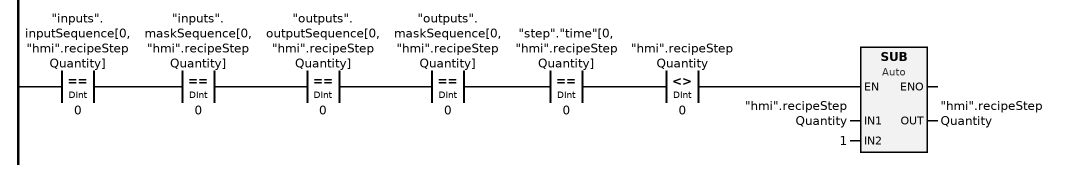
   RUNG wire#powerrail
      { S7_Templates := "SrcType := DInt" } NE_Contact(in1 := "inputs".inputSequence[0, 25], in2 := 0)
      wire#w1
      Move(in := 25, out1 => "hmi".recipeStepQuantity)
   END_RUNG
   RUNG wire#powerrail
      { S7_Templates := "SrcType := DInt" } NE_Contact(in1 := "inputs".maskSequence[0, 25], in2 := 0)
   END_RUNG wire#w1
   RUNG wire#powerrail
      { S7_Templates := "SrcType := DInt" } NE_Contact(in1 := "outputs".outputSequence[0, 25], in2 := 0)
   END_RUNG wire#w1
   RUNG wire#powerrail
      { S7_Templates := "SrcType := DInt" } NE_Contact(in1 := "outputs".maskSequence[0, 25], in2 := 0)
   END_RUNG wire#w1
   RUNG wire#powerrail
      { S7_Templates := "SrcType := DInt" } NE_Contact(in1 := "step"."time"[0, 25], in2 := 0)
   END_RUNG wire#w1
   RUNG wire#powerrail
      { S7_Templates := "SrcType := DInt" } LT_Contact(in1 := "hmi".recipeStepQuantity, in2 := 25)
      wire#w2
      { S7_Templates := "SrcType := DInt" } NE_Contact(in1 := "inputs".inputSequence[0, 24], in2 := 0)
      wire#w3
      Move(in := 24, out1 => "hmi".recipeStepQuantity)
   END_RUNG
   RUNG wire#w2
      { S7_Templates := "SrcType := DInt" } NE_Contact(in1 := "inputs".maskSequence[0, 24], in2 := 0)
   END_RUNG wire#w3
   RUNG wire#w2
      { S7_Templates := "SrcType := DInt" } NE_Contact(in1 := "outputs".outputSequence[0, 24], in2 := 0)
   END_RUNG wire#w3
   RUNG wire#w2
      { S7_Templates := "SrcType := DInt" } NE_Contact(in1 := "outputs".maskSequence[0, 24], in2 := 0)
   END_RUNG wire#w3
   RUNG wire#w2
      { S7_Templates := "SrcType := DInt" } NE_Contact(in1 := "step"."time"[0, 24], in2 := 0)
   END_RUNG wire#w3
   RUNG wire#powerrail
      { S7_Templates := "SrcType := DInt" } LT_Contact(in1 := "hmi".recipeStepQuantity, in2 := 24)
      wire#w4
      { S7_Templates := "SrcType := DInt" } NE_Contact(in1 := "inputs".inputSequence[0, 23], in2 := 0)
      wire#w5
      Move(in := 23, out1 => "hmi".recipeStepQuantity)
   END_RUNG
   RUNG wire#w4
      { S7_Templates := "SrcType := DInt" } NE_Contact(in1 := "inputs".maskSequence[0, 23], in2 := 0)
   END_RUNG wire#w5
   RUNG wire#w4
      { S7_Templates := "SrcType := DInt" } NE_Contact(in1 := "outputs".outputSequence[0, 23], in2 := 0)
   END_RUNG wire#w5
   RUNG wire#w4
      { S7_Templates := "SrcType := DInt" } NE_Contact(in1 := "outputs".maskSequence[0, 23], in2 := 0)
   END_RUNG wire#w5
   RUNG wire#w4
      { S7_Templates := "SrcType := DInt" } NE_Contact(in1 := "step"."time"[0, 23], in2 := 0)
   END_RUNG wire#w5
   RUNG wire#powerrail
      { S7_Templates := "SrcType := DInt" } LT_Contact(in1 := "hmi".recipeStepQuantity, in2 := 23)
      wire#w6
      { S7_Templates := "SrcType := DInt" } NE_Contact(in1 := "inputs".inputSequence[0, 22], in2 := 0)
      wire#w7
      Move(in := 22, out1 => "hmi".recipeStepQuantity)
   END_RUNG
   RUNG wire#w6
      { S7_Templates := "SrcType := DInt" } NE_Contact(in1 := "inputs".maskSequence[0, 22], in2 := 0)
   END_RUNG wire#w7
   RUNG wire#w6
      { S7_Templates := "SrcType := DInt" } NE_Contact(in1 := "outputs".outputSequence[0, 22], in2 := 0)
   END_RUNG wire#w7
   RUNG wire#w6
      { S7_Templates := "SrcType := DInt" } NE_Contact(in1 := "outputs".maskSequence[0, 22], in2 := 0)
   END_RUNG wire#w7
   RUNG wire#w6
      { S7_Templates := "SrcType := DInt" } NE_Contact(in1 := "step"."time"[0, 22], in2 := 0)
   END_RUNG wire#w7
   RUNG wire#powerrail
      { S7_Templates := "SrcType := DInt" } LT_Contact(in1 := "hmi".recipeStepQuantity, in2 := 22)
      wire#w8
      { S7_Templates := "SrcType := DInt" } NE_Contact(in1 := "inputs".inputSequence[0, 21], in2 := 0)
      wire#w9
      Move(in := 21, out1 => "hmi".recipeStepQuantity)
   END_RUNG
   RUNG wire#w8
      { S7_Templates := "SrcType := DInt" } NE_Contact(in1 := "inputs".maskSequence[0, 21], in2 := 0)
   END_RUNG wire#w9
   RUNG wire#w8
      { S7_Templates := "SrcType := DInt" } NE_Contact(in1 := "outputs".outputSequence[0, 21], in2 := 0)
   END_RUNG wire#w9
   RUNG wire#w8
      { S7_Templates := "SrcType := DInt" } NE_Contact(in1 := "outputs".maskSequence[0, 21], in2 := 0)
   END_RUNG wire#w9
   RUNG wire#w8
      { S7_Templates := "SrcType := DInt" } NE_Contact(in1 := "step"."time"[0, 21], in2 := 0)
   END_RUNG wire#w9
   RUNG wire#powerrail
      { S7_Templates := "SrcType := DInt" } LT_Contact(in1 := "hmi".recipeStepQuantity, in2 := 21)
      wire#w10
      { S7_Templates := "SrcType := DInt" } NE_Contact(in1 := "inputs".inputSequence[0, 20], in2 := 0)
      wire#w11
      Move(in := 20, out1 => "hmi".recipeStepQuantity)
   END_RUNG
   RUNG wire#w10
      { S7_Templates := "SrcType := DInt" } NE_Contact(in1 := "inputs".maskSequence[0, 20], in2 := 0)
   END_RUNG wire#w11
   RUNG wire#w10
      { S7_Templates := "SrcType := DInt" } NE_Contact(in1 := "outputs".outputSequence[0, 20], in2 := 0)
   END_RUNG wire#w11
   RUNG wire#w10
      { S7_Templates := "SrcType := DInt" } NE_Contact(in1 := "outputs".maskSequence[0, 20], in2 := 0)
   END_RUNG wire#w11
   RUNG wire#w10
      { S7_Templates := "SrcType := DInt" } NE_Contact(in1 := "step"."time"[0, 20], in2 := 0)
   END_RUNG wire#w11
   RUNG wire#powerrail
      { S7_Templates := "SrcType := DInt" } LT_Contact(in1 := "hmi".recipeStepQuantity, in2 := 20)
      wire#w12
      { S7_Templates := "SrcType := DInt" } NE_Contact(in1 := "inputs".inputSequence[0, 19], in2 := 0)
      wire#w13
      Move(in := 19, out1 => "hmi".recipeStepQuantity)
   END_RUNG
   RUNG wire#w12
      { S7_Templates := "SrcType := DInt" } NE_Contact(in1 := "inputs".maskSequence[0, 19], in2 := 0)
   END_RUNG wire#w13
   RUNG wire#w12
      { S7_Templates := "SrcType := DInt" } NE_Contact(in1 := "outputs".outputSequence[0, 19], in2 := 0)
   END_RUNG wire#w13
   RUNG wire#w12
      { S7_Templates := "SrcType := DInt" } NE_Contact(in1 := "outputs".maskSequence[0, 19], in2 := 0)
   END_RUNG wire#w13
   RUNG wire#w12
      { S7_Templates := "SrcType := DInt" } NE_Contact(in1 := "step"."time"[0, 19], in2 := 0)
   END_RUNG wire#w13
   RUNG wire#powerrail
      { S7_Templates := "SrcType := DInt" } LT_Contact(in1 := "hmi".recipeStepQuantity, in2 := 19)
      wire#w14
      { S7_Templates := "SrcType := DInt" } NE_Contact(in1 := "inputs".inputSequence[0, 18], in2 := 0)
      wire#w15
      Move(in := 18, out1 => "hmi".recipeStepQuantity)
   END_RUNG
   RUNG wire#w14
      { S7_Templates := "SrcType := DInt" } NE_Contact(in1 := "inputs".maskSequence[0, 18], in2 := 0)
   END_RUNG wire#w15
   RUNG wire#w14
      { S7_Templates := "SrcType := DInt" } NE_Contact(in1 := "outputs".outputSequence[0, 18], in2 := 0)
   END_RUNG wire#w15
   RUNG wire#w14
      { S7_Templates := "SrcType := DInt" } NE_Contact(in1 := "outputs".maskSequence[0, 18], in2 := 0)
   END_RUNG wire#w15
   RUNG wire#w14
      { S7_Templates := "SrcType := DInt" } NE_Contact(in1 := "step"."time"[0, 18], in2 := 0)
   END_RUNG wire#w15
   RUNG wire#powerrail
      { S7_Templates := "SrcType := DInt" } LT_Contact(in1 := "hmi".recipeStepQuantity, in2 := 18)
      wire#w16
      { S7_Templates := "SrcType := DInt" } NE_Contact(in1 := "inputs".inputSequence[0, 17], in2 := 0)
      wire#w17
      Move(in := 17, out1 => "hmi".recipeStepQuantity)
   END_RUNG
   RUNG wire#w16
      { S7_Templates := "SrcType := DInt" } NE_Contact(in1 := "inputs".maskSequence[0, 17], in2 := 0)
   END_RUNG wire#w17
   RUNG wire#w16
      { S7_Templates := "SrcType := DInt" } NE_Contact(in1 := "outputs".outputSequence[0, 17], in2 := 0)
   END_RUNG wire#w17
   RUNG wire#w16
      { S7_Templates := "SrcType := DInt" } NE_Contact(in1 := "outputs".maskSequence[0, 17], in2 := 0)
   END_RUNG wire#w17
   RUNG wire#w16
      { S7_Templates := "SrcType := DInt" } NE_Contact(in1 := "step"."time"[0, 17], in2 := 0)
   END_RUNG wire#w17
   RUNG wire#powerrail
      { S7_Templates := "SrcType := DInt" } LT_Contact(in1 := "hmi".recipeStepQuantity, in2 := 17)
      wire#w18
      { S7_Templates := "SrcType := DInt" } NE_Contact(in1 := "inputs".inputSequence[0, 16], in2 := 0)
      wire#w19
      Move(in := 16, out1 => "hmi".recipeStepQuantity)
   END_RUNG
   RUNG wire#w18
      { S7_Templates := "SrcType := DInt" } NE_Contact(in1 := "inputs".maskSequence[0, 16], in2 := 0)
   END_RUNG wire#w19
   RUNG wire#w18
      { S7_Templates := "SrcType := DInt" } NE_Contact(in1 := "outputs".outputSequence[0, 16], in2 := 0)
   END_RUNG wire#w19
   RUNG wire#w18
      { S7_Templates := "SrcType := DInt" } NE_Contact(in1 := "outputs".maskSequence[0, 16], in2 := 0)
   END_RUNG wire#w19
   RUNG wire#w18
      { S7_Templates := "SrcType := DInt" } NE_Contact(in1 := "step"."time"[0, 16], in2 := 0)
   END_RUNG wire#w19
   RUNG wire#powerrail
      { S7_Templates := "SrcType := DInt" } LT_Contact(in1 := "hmi".recipeStepQuantity, in2 := 16)
      wire#w20
      { S7_Templates := "SrcType := DInt" } NE_Contact(in1 := "inputs".inputSequence[0, 15], in2 := 0)
      wire#w21
      Move(in := 15, out1 => "hmi".recipeStepQuantity)
   END_RUNG
   RUNG wire#w20
      { S7_Templates := "SrcType := DInt" } NE_Contact(in1 := "inputs".maskSequence[0, 15], in2 := 0)
   END_RUNG wire#w21
   RUNG wire#w20
      { S7_Templates := "SrcType := DInt" } NE_Contact(in1 := "outputs".outputSequence[0, 15], in2 := 0)
   END_RUNG wire#w21
   RUNG wire#w20
      { S7_Templates := "SrcType := DInt" } NE_Contact(in1 := "outputs".maskSequence[0, 15], in2 := 0)
   END_RUNG wire#w21
   RUNG wire#w20
      { S7_Templates := "SrcType := DInt" } NE_Contact(in1 := "step"."time"[0, 15], in2 := 0)
   END_RUNG wire#w21
   RUNG wire#powerrail
      { S7_Templates := "SrcType := DInt" } LT_Contact(in1 := "hmi".recipeStepQuantity, in2 := 15)
      wire#w22
      { S7_Templates := "SrcType := DInt" } NE_Contact(in1 := "inputs".inputSequence[0, 14], in2 := 0)
      wire#w23
      Move(in := 14, out1 => "hmi".recipeStepQuantity)
   END_RUNG
   RUNG wire#w22
      { S7_Templates := "SrcType := DInt" } NE_Contact(in1 := "inputs".maskSequence[0, 14], in2 := 0)
   END_RUNG wire#w23
   RUNG wire#w22
      { S7_Templates := "SrcType := DInt" } NE_Contact(in1 := "outputs".outputSequence[0, 14], in2 := 0)
   END_RUNG wire#w23
   RUNG wire#w22
      { S7_Templates := "SrcType := DInt" } NE_Contact(in1 := "outputs".maskSequence[0, 14], in2 := 0)
   END_RUNG wire#w23
   RUNG wire#w22
      { S7_Templates := "SrcType := DInt" } NE_Contact(in1 := "step"."time"[0, 14], in2 := 0)
   END_RUNG wire#w23
   RUNG wire#powerrail
      { S7_Templates := "SrcType := DInt" } LT_Contact(in1 := "hmi".recipeStepQuantity, in2 := 14)
      wire#w24
      { S7_Templates := "SrcType := DInt" } NE_Contact(in1 := "inputs".inputSequence[0, 13], in2 := 0)
      wire#w25
      Move(in := 13, out1 => "hmi".recipeStepQuantity)
   END_RUNG
   RUNG wire#w24
      { S7_Templates := "SrcType := DInt" } NE_Contact(in1 := "inputs".maskSequence[0, 13], in2 := 0)
   END_RUNG wire#w25
   RUNG wire#w24
      { S7_Templates := "SrcType := DInt" } NE_Contact(in1 := "outputs".outputSequence[0, 13], in2 := 0)
   END_RUNG wire#w25
   RUNG wire#w24
      { S7_Templates := "SrcType := DInt" } NE_Contact(in1 := "outputs".maskSequence[0, 13], in2 := 0)
   END_RUNG wire#w25
   RUNG wire#w24
      { S7_Templates := "SrcType := DInt" } NE_Contact(in1 := "step"."time"[0, 13], in2 := 0)
   END_RUNG wire#w25
   RUNG wire#powerrail
      { S7_Templates := "SrcType := DInt" } LT_Contact(in1 := "hmi".recipeStepQuantity, in2 := 13)
      wire#w26
      { S7_Templates := "SrcType := DInt" } NE_Contact(in1 := "inputs".inputSequence[0, 12], in2 := 0)
      wire#w27
      Move(in := 12, out1 => "hmi".recipeStepQuantity)
   END_RUNG
   RUNG wire#w26
      { S7_Templates := "SrcType := DInt" } NE_Contact(in1 := "inputs".maskSequence[0, 12], in2 := 0)
   END_RUNG wire#w27
   RUNG wire#w26
      { S7_Templates := "SrcType := DInt" } NE_Contact(in1 := "outputs".outputSequence[0, 12], in2 := 0)
   END_RUNG wire#w27
   RUNG wire#w26
      { S7_Templates := "SrcType := DInt" } NE_Contact(in1 := "outputs".maskSequence[0, 12], in2 := 0)
   END_RUNG wire#w27
   RUNG wire#w26
      { S7_Templates := "SrcType := DInt" } NE_Contact(in1 := "step"."time"[0, 12], in2 := 0)
   END_RUNG wire#w27
   RUNG wire#powerrail
      { S7_Templates := "SrcType := DInt" } LT_Contact(in1 := "hmi".recipeStepQuantity, in2 := 12)
      wire#w28
      { S7_Templates := "SrcType := DInt" } NE_Contact(in1 := "inputs".inputSequence[0, 11], in2 := 0)
      wire#w29
      Move(in := 11, out1 => "hmi".recipeStepQuantity)
   END_RUNG
   RUNG wire#w28
      { S7_Templates := "SrcType := DInt" } NE_Contact(in1 := "inputs".maskSequence[0, 11], in2 := 0)
   END_RUNG wire#w29
   RUNG wire#w28
      { S7_Templates := "SrcType := DInt" } NE_Contact(in1 := "outputs".outputSequence[0, 11], in2 := 0)
   END_RUNG wire#w29
   RUNG wire#w28
      { S7_Templates := "SrcType := DInt" } NE_Contact(in1 := "outputs".maskSequence[0, 11], in2 := 0)
   END_RUNG wire#w29
   RUNG wire#w28
      { S7_Templates := "SrcType := DInt" } NE_Contact(in1 := "step"."time"[0, 11], in2 := 0)
   END_RUNG wire#w29
   RUNG wire#powerrail
      { S7_Templates := "SrcType := DInt" } LT_Contact(in1 := "hmi".recipeStepQuantity, in2 := 11)
      wire#w30
      { S7_Templates := "SrcType := DInt" } NE_Contact(in1 := "inputs".inputSequence[0, 10], in2 := 0)
      wire#w31
      Move(in := 10, out1 => "hmi".recipeStepQuantity)
   END_RUNG
   RUNG wire#w30
      { S7_Templates := "SrcType := DInt" } NE_Contact(in1 := "inputs".maskSequence[0, 10], in2 := 0)
   END_RUNG wire#w31
   RUNG wire#w30
      { S7_Templates := "SrcType := DInt" } NE_Contact(in1 := "outputs".outputSequence[0, 10], in2 := 0)
   END_RUNG wire#w31
   RUNG wire#w30
      { S7_Templates := "SrcType := DInt" } NE_Contact(in1 := "outputs".maskSequence[0, 10], in2 := 0)
   END_RUNG wire#w31
   RUNG wire#w30
      { S7_Templates := "SrcType := DInt" } NE_Contact(in1 := "step"."time"[0, 10], in2 := 0)
   END_RUNG wire#w31
   RUNG wire#powerrail
      { S7_Templates := "SrcType := DInt" } LT_Contact(in1 := "hmi".recipeStepQuantity, in2 := 10)
      wire#w32
      { S7_Templates := "SrcType := DInt" } NE_Contact(in1 := "inputs".inputSequence[0, 9], in2 := 0)
      wire#w33
      Move(in := 9, out1 => "hmi".recipeStepQuantity)
   END_RUNG
   RUNG wire#w32
      { S7_Templates := "SrcType := DInt" } NE_Contact(in1 := "inputs".maskSequence[0, 9], in2 := 0)
   END_RUNG wire#w33
   RUNG wire#w32
      { S7_Templates := "SrcType := DInt" } NE_Contact(in1 := "outputs".outputSequence[0, 9], in2 := 0)
   END_RUNG wire#w33
   RUNG wire#w32
      { S7_Templates := "SrcType := DInt" } NE_Contact(in1 := "outputs".maskSequence[0, 9], in2 := 0)
   END_RUNG wire#w33
   RUNG wire#w32
      { S7_Templates := "SrcType := DInt" } NE_Contact(in1 := "step"."time"[0, 9], in2 := 0)
   END_RUNG wire#w33
   RUNG wire#powerrail
      { S7_Templates := "SrcType := DInt" } LT_Contact(in1 := "hmi".recipeStepQuantity, in2 := 9)
      wire#w34
      { S7_Templates := "SrcType := DInt" } NE_Contact(in1 := "inputs".inputSequence[0, 8], in2 := 0)
      wire#w35
      Move(in := 8, out1 => "hmi".recipeStepQuantity)
   END_RUNG
   RUNG wire#w34
      { S7_Templates := "SrcType := DInt" } NE_Contact(in1 := "inputs".maskSequence[0, 8], in2 := 0)
   END_RUNG wire#w35
   RUNG wire#w34
      { S7_Templates := "SrcType := DInt" } NE_Contact(in1 := "outputs".outputSequence[0, 8], in2 := 0)
   END_RUNG wire#w35
   RUNG wire#w34
      { S7_Templates := "SrcType := DInt" } NE_Contact(in1 := "outputs".maskSequence[0, 8], in2 := 0)
   END_RUNG wire#w35
   RUNG wire#w34
      { S7_Templates := "SrcType := DInt" } NE_Contact(in1 := "step"."time"[0, 8], in2 := 0)
   END_RUNG wire#w35
   RUNG wire#powerrail
      { S7_Templates := "SrcType := DInt" } LT_Contact(in1 := "hmi".recipeStepQuantity, in2 := 8)
      wire#w36
      { S7_Templates := "SrcType := DInt" } NE_Contact(in1 := "inputs".inputSequence[0, 7], in2 := 0)
      wire#w37
      Move(in := 7, out1 => "hmi".recipeStepQuantity)
   END_RUNG
   RUNG wire#w36
      { S7_Templates := "SrcType := DInt" } NE_Contact(in1 := "inputs".maskSequence[0, 7], in2 := 0)
   END_RUNG wire#w37
   RUNG wire#w36
      { S7_Templates := "SrcType := DInt" } NE_Contact(in1 := "outputs".outputSequence[0, 7], in2 := 0)
   END_RUNG wire#w37
   RUNG wire#w36
      { S7_Templates := "SrcType := DInt" } NE_Contact(in1 := "outputs".maskSequence[0, 7], in2 := 0)
   END_RUNG wire#w37
   RUNG wire#w36
      { S7_Templates := "SrcType := DInt" } NE_Contact(in1 := "step"."time"[0, 7], in2 := 0)
   END_RUNG wire#w37
   RUNG wire#powerrail
      { S7_Templates := "SrcType := DInt" } LT_Contact(in1 := "hmi".recipeStepQuantity, in2 := 7)
      wire#w38
      { S7_Templates := "SrcType := DInt" } NE_Contact(in1 := "inputs".inputSequence[0, 6], in2 := 0)
      wire#w39
      Move(in := 6, out1 => "hmi".recipeStepQuantity)
   END_RUNG
   RUNG wire#w38
      { S7_Templates := "SrcType := DInt" } NE_Contact(in1 := "inputs".maskSequence[0, 6], in2 := 0)
   END_RUNG wire#w39
   RUNG wire#w38
      { S7_Templates := "SrcType := DInt" } NE_Contact(in1 := "outputs".outputSequence[0, 6], in2 := 0)
   END_RUNG wire#w39
   RUNG wire#w38
      { S7_Templates := "SrcType := DInt" } NE_Contact(in1 := "outputs".maskSequence[0, 6], in2 := 0)
   END_RUNG wire#w39
   RUNG wire#w38
      { S7_Templates := "SrcType := DInt" } NE_Contact(in1 := "step"."time"[0, 6], in2 := 0)
   END_RUNG wire#w39
   RUNG wire#powerrail
      { S7_Templates := "SrcType := DInt" } LT_Contact(in1 := "hmi".recipeStepQuantity, in2 := 6)
      wire#w40
      { S7_Templates := "SrcType := DInt" } NE_Contact(in1 := "inputs".inputSequence[0, 5], in2 := 0)
      wire#w41
      Move(in := 5, out1 => "hmi".recipeStepQuantity)
   END_RUNG
   RUNG wire#w40
      { S7_Templates := "SrcType := DInt" } NE_Contact(in1 := "inputs".maskSequence[0, 5], in2 := 0)
   END_RUNG wire#w41
   RUNG wire#w40
      { S7_Templates := "SrcType := DInt" } NE_Contact(in1 := "outputs".outputSequence[0, 5], in2 := 0)
   END_RUNG wire#w41
   RUNG wire#w40
      { S7_Templates := "SrcType := DInt" } NE_Contact(in1 := "outputs".maskSequence[0, 5], in2 := 0)
   END_RUNG wire#w41
   RUNG wire#w40
      { S7_Templates := "SrcType := DInt" } NE_Contact(in1 := "step"."time"[0, 5], in2 := 0)
   END_RUNG wire#w41
   RUNG wire#powerrail
      { S7_Templates := "SrcType := DInt" } LT_Contact(in1 := "hmi".recipeStepQuantity, in2 := 5)
      wire#w42
      { S7_Templates := "SrcType := DInt" } NE_Contact(in1 := "inputs".inputSequence[0, 4], in2 := 0)
      wire#w43
      Move(in := 4, out1 => "hmi".recipeStepQuantity)
   END_RUNG
   RUNG wire#w42
      { S7_Templates := "SrcType := DInt" } NE_Contact(in1 := "inputs".maskSequence[0, 4], in2 := 0)
   END_RUNG wire#w43
   RUNG wire#w42
      { S7_Templates := "SrcType := DInt" } NE_Contact(in1 := "outputs".outputSequence[0, 4], in2 := 0)
   END_RUNG wire#w43
   RUNG wire#w42
      { S7_Templates := "SrcType := DInt" } NE_Contact(in1 := "outputs".maskSequence[0, 4], in2 := 0)
   END_RUNG wire#w43
   RUNG wire#w42
      { S7_Templates := "SrcType := DInt" } NE_Contact(in1 := "step"."time"[0, 4], in2 := 0)
   END_RUNG wire#w43
   RUNG wire#powerrail
      { S7_Templates := "SrcType := DInt" } LT_Contact(in1 := "hmi".recipeStepQuantity, in2 := 4)
      wire#w44
      { S7_Templates := "SrcType := DInt" } NE_Contact(in1 := "inputs".inputSequence[0, 3], in2 := 0)
      wire#w45
      Move(in := 3, out1 => "hmi".recipeStepQuantity)
   END_RUNG
   RUNG wire#w44
      { S7_Templates := "SrcType := DInt" } NE_Contact(in1 := "inputs".maskSequence[0, 3], in2 := 0)
   END_RUNG wire#w45
   RUNG wire#w44
      { S7_Templates := "SrcType := DInt" } NE_Contact(in1 := "outputs".outputSequence[0, 3], in2 := 0)
   END_RUNG wire#w45
   RUNG wire#w44
      { S7_Templates := "SrcType := DInt" } NE_Contact(in1 := "outputs".maskSequence[0, 3], in2 := 0)
   END_RUNG wire#w45
   RUNG wire#w44
      { S7_Templates := "SrcType := DInt" } NE_Contact(in1 := "step"."time"[0, 3], in2 := 0)
   END_RUNG wire#w45
   RUNG wire#powerrail
      { S7_Templates := "SrcType := DInt" } LT_Contact(in1 := "hmi".recipeStepQuantity, in2 := 3)
      wire#w46
      { S7_Templates := "SrcType := DInt" } NE_Contact(in1 := "inputs".inputSequence[0, 2], in2 := 0)
      wire#w47
      Move(in := 2, out1 => "hmi".recipeStepQuantity)
   END_RUNG
   RUNG wire#w46
      { S7_Templates := "SrcType := DInt" } NE_Contact(in1 := "inputs".maskSequence[0, 2], in2 := 0)
   END_RUNG wire#w47
   RUNG wire#w46
      { S7_Templates := "SrcType := DInt" } NE_Contact(in1 := "outputs".outputSequence[0, 2], in2 := 0)
   END_RUNG wire#w47
   RUNG wire#w46
      { S7_Templates := "SrcType := DInt" } NE_Contact(in1 := "outputs".maskSequence[0, 2], in2 := 0)
   END_RUNG wire#w47
   RUNG wire#w46
      { S7_Templates := "SrcType := DInt" } NE_Contact(in1 := "step"."time"[0, 2], in2 := 0)
   END_RUNG wire#w47
   RUNG wire#powerrail
      { S7_Templates := "SrcType := DInt" } LT_Contact(in1 := "hmi".recipeStepQuantity, in2 := 2)
      wire#w48
      { S7_Templates := "SrcType := DInt" } NE_Contact(in1 := "inputs".inputSequence[0, 1], in2 := 0)
      wire#w49
      Move(in := 1, out1 => "hmi".recipeStepQuantity)
   END_RUNG
   RUNG wire#w48
      { S7_Templates := "SrcType := DInt" } NE_Contact(in1 := "inputs".maskSequence[0, 1], in2 := 0)
   END_RUNG wire#w49
   RUNG wire#w48
      { S7_Templates := "SrcType := DInt" } NE_Contact(in1 := "outputs".outputSequence[0, 1], in2 := 0)
   END_RUNG wire#w49
   RUNG wire#w48
      { S7_Templates := "SrcType := DInt" } NE_Contact(in1 := "outputs".maskSequence[0, 1], in2 := 0)
   END_RUNG wire#w49
   RUNG wire#w48
      { S7_Templates := "SrcType := DInt" } NE_Contact(in1 := "step"."time"[0, 1], in2 := 0)
   END_RUNG wire#w49
   RUNG wire#powerrail
      { S7_Templates := "SrcType := DInt" } LT_Contact(in1 := "hmi".recipeStepQuantity, in2 := 1)
      Move(in := 0, out1 => "hmi".recipeStepQuantity)
   END_RUNG
   RUNG wire#powerrail
      { S7_Templates := "SrcType := DInt" } EQ_Contact(in1 := "inputs".inputSequence[0, "hmi".recipeStepQuantity], in2 := 0)
      { S7_Templates := "SrcType := DInt" } EQ_Contact(in1 := "inputs".maskSequence[0, "hmi".recipeStepQuantity], in2 := 0)
      { S7_Templates := "SrcType := DInt" } EQ_Contact(in1 := "outputs".outputSequence[0, "hmi".recipeStepQuantity], in2 := 0)
      { S7_Templates := "SrcType := DInt" } EQ_Contact(in1 := "outputs".maskSequence[0, "hmi".recipeStepQuantity], in2 := 0)
      { S7_Templates := "SrcType := DInt" } EQ_Contact(in1 := "step"."time"[0, "hmi".recipeStepQuantity], in2 := 0)
      { S7_Templates := "SrcType := DInt" } NE_Contact(in1 := "hmi".recipeStepQuantity, in2 := 0)
      Sub(in1 := "hmi".recipeStepQuantity, in2 := 1, out => "hmi".recipeStepQuantity)
   END_RUNG
   // the same network as SCL:
   IF ("inputs".inputSequence[0, 25] <> 0) OR ("inputs".maskSequence[0, 25] <> 0) OR ("outputs".outputSequence[0, 25] <> 0) OR ("outputs".maskSequence[0, 25] <> 0) OR ("step"."time"[0, 25] <> 0) THEN
       "hmi".recipeStepQuantity := 25;
   END_IF;
   IF ("hmi".recipeStepQuantity < 25) AND (("inputs".inputSequence[0, 24] <> 0) OR ("inputs".maskSequence[0, 24] <> 0) OR ("outputs".outputSequence[0, 24] <> 0) OR ("outputs".maskSequence[0, 24] <> 0) OR ("step"."time"[0, 24] <> 0)) THEN
       "hmi".recipeStepQuantity := 24;
   END_IF;
   IF ("hmi".recipeStepQuantity < 24) AND (("inputs".inputSequence[0, 23] <> 0) OR ("inputs".maskSequence[0, 23] <> 0) OR ("outputs".outputSequence[0, 23] <> 0) OR ("outputs".maskSequence[0, 23] <> 0) OR ("step"."time"[0, 23] <> 0)) THEN
       "hmi".recipeStepQuantity := 23;
   END_IF;
   IF ("hmi".recipeStepQuantity < 23) AND (("inputs".inputSequence[0, 22] <> 0) OR ("inputs".maskSequence[0, 22] <> 0) OR ("outputs".outputSequence[0, 22] <> 0) OR ("outputs".maskSequence[0, 22] <> 0) OR ("step"."time"[0, 22] <> 0)) THEN
       "hmi".recipeStepQuantity := 22;
   END_IF;
   IF ("hmi".recipeStepQuantity < 22) AND (("inputs".inputSequence[0, 21] <> 0) OR ("inputs".maskSequence[0, 21] <> 0) OR ("outputs".outputSequence[0, 21] <> 0) OR ("outputs".maskSequence[0, 21] <> 0) OR ("step"."time"[0, 21] <> 0)) THEN
       "hmi".recipeStepQuantity := 21;
   END_IF;
   IF ("hmi".recipeStepQuantity < 21) AND (("inputs".inputSequence[0, 20] <> 0) OR ("inputs".maskSequence[0, 20] <> 0) OR ("outputs".outputSequence[0, 20] <> 0) OR ("outputs".maskSequence[0, 20] <> 0) OR ("step"."time"[0, 20] <> 0)) THEN
       "hmi".recipeStepQuantity := 20;
   END_IF;
   IF ("hmi".recipeStepQuantity < 20) AND (("inputs".inputSequence[0, 19] <> 0) OR ("inputs".maskSequence[0, 19] <> 0) OR ("outputs".outputSequence[0, 19] <> 0) OR ("outputs".maskSequence[0, 19] <> 0) OR ("step"."time"[0, 19] <> 0)) THEN
       "hmi".recipeStepQuantity := 19;
   END_IF;
   IF ("hmi".recipeStepQuantity < 19) AND (("inputs".inputSequence[0, 18] <> 0) OR ("inputs".maskSequence[0, 18] <> 0) OR ("outputs".outputSequence[0, 18] <> 0) OR ("outputs".maskSequence[0, 18] <> 0) OR ("step"."time"[0, 18] <> 0)) THEN
       "hmi".recipeStepQuantity := 18;
   END_IF;
   IF ("hmi".recipeStepQuantity < 18) AND (("inputs".inputSequence[0, 17] <> 0) OR ("inputs".maskSequence[0, 17] <> 0) OR ("outputs".outputSequence[0, 17] <> 0) OR ("outputs".maskSequence[0, 17] <> 0) OR ("step"."time"[0, 17] <> 0)) THEN
       "hmi".recipeStepQuantity := 17;
   END_IF;
   IF ("hmi".recipeStepQuantity < 17) AND (("inputs".inputSequence[0, 16] <> 0) OR ("inputs".maskSequence[0, 16] <> 0) OR ("outputs".outputSequence[0, 16] <> 0) OR ("outputs".maskSequence[0, 16] <> 0) OR ("step"."time"[0, 16] <> 0)) THEN
       "hmi".recipeStepQuantity := 16;
   END_IF;
   IF ("hmi".recipeStepQuantity < 16) AND (("inputs".inputSequence[0, 15] <> 0) OR ("inputs".maskSequence[0, 15] <> 0) OR ("outputs".outputSequence[0, 15] <> 0) OR ("outputs".maskSequence[0, 15] <> 0) OR ("step"."time"[0, 15] <> 0)) THEN
       "hmi".recipeStepQuantity := 15;
   END_IF;
   IF ("hmi".recipeStepQuantity < 15) AND (("inputs".inputSequence[0, 14] <> 0) OR ("inputs".maskSequence[0, 14] <> 0) OR ("outputs".outputSequence[0, 14] <> 0) OR ("outputs".maskSequence[0, 14] <> 0) OR ("step"."time"[0, 14] <> 0)) THEN
       "hmi".recipeStepQuantity := 14;
   END_IF;
   IF ("hmi".recipeStepQuantity < 14) AND (("inputs".inputSequence[0, 13] <> 0) OR ("inputs".maskSequence[0, 13] <> 0) OR ("outputs".outputSequence[0, 13] <> 0) OR ("outputs".maskSequence[0, 13] <> 0) OR ("step"."time"[0, 13] <> 0)) THEN
       "hmi".recipeStepQuantity := 13;
   END_IF;
   IF ("hmi".recipeStepQuantity < 13) AND (("inputs".inputSequence[0, 12] <> 0) OR ("inputs".maskSequence[0, 12] <> 0) OR ("outputs".outputSequence[0, 12] <> 0) OR ("outputs".maskSequence[0, 12] <> 0) OR ("step"."time"[0, 12] <> 0)) THEN
       "hmi".recipeStepQuantity := 12;
   END_IF;
   IF ("hmi".recipeStepQuantity < 12) AND (("inputs".inputSequence[0, 11] <> 0) OR ("inputs".maskSequence[0, 11] <> 0) OR ("outputs".outputSequence[0, 11] <> 0) OR ("outputs".maskSequence[0, 11] <> 0) OR ("step"."time"[0, 11] <> 0)) THEN
       "hmi".recipeStepQuantity := 11;
   END_IF;
   IF ("hmi".recipeStepQuantity < 11) AND (("inputs".inputSequence[0, 10] <> 0) OR ("inputs".maskSequence[0, 10] <> 0) OR ("outputs".outputSequence[0, 10] <> 0) OR ("outputs".maskSequence[0, 10] <> 0) OR ("step"."time"[0, 10] <> 0)) THEN
       "hmi".recipeStepQuantity := 10;
   END_IF;
   IF ("hmi".recipeStepQuantity < 10) AND (("inputs".inputSequence[0, 9] <> 0) OR ("inputs".maskSequence[0, 9] <> 0) OR ("outputs".outputSequence[0, 9] <> 0) OR ("outputs".maskSequence[0, 9] <> 0) OR ("step"."time"[0, 9] <> 0)) THEN
       "hmi".recipeStepQuantity := 9;
   END_IF;
   IF ("hmi".recipeStepQuantity < 9) AND (("inputs".inputSequence[0, 8] <> 0) OR ("inputs".maskSequence[0, 8] <> 0) OR ("outputs".outputSequence[0, 8] <> 0) OR ("outputs".maskSequence[0, 8] <> 0) OR ("step"."time"[0, 8] <> 0)) THEN
       "hmi".recipeStepQuantity := 8;
   END_IF;
   IF ("hmi".recipeStepQuantity < 8) AND (("inputs".inputSequence[0, 7] <> 0) OR ("inputs".maskSequence[0, 7] <> 0) OR ("outputs".outputSequence[0, 7] <> 0) OR ("outputs".maskSequence[0, 7] <> 0) OR ("step"."time"[0, 7] <> 0)) THEN
       "hmi".recipeStepQuantity := 7;
   END_IF;
   IF ("hmi".recipeStepQuantity < 7) AND (("inputs".inputSequence[0, 6] <> 0) OR ("inputs".maskSequence[0, 6] <> 0) OR ("outputs".outputSequence[0, 6] <> 0) OR ("outputs".maskSequence[0, 6] <> 0) OR ("step"."time"[0, 6] <> 0)) THEN
       "hmi".recipeStepQuantity := 6;
   END_IF;
   IF ("hmi".recipeStepQuantity < 6) AND (("inputs".inputSequence[0, 5] <> 0) OR ("inputs".maskSequence[0, 5] <> 0) OR ("outputs".outputSequence[0, 5] <> 0) OR ("outputs".maskSequence[0, 5] <> 0) OR ("step"."time"[0, 5] <> 0)) THEN
       "hmi".recipeStepQuantity := 5;
   END_IF;
   IF ("hmi".recipeStepQuantity < 5) AND (("inputs".inputSequence[0, 4] <> 0) OR ("inputs".maskSequence[0, 4] <> 0) OR ("outputs".outputSequence[0, 4] <> 0) OR ("outputs".maskSequence[0, 4] <> 0) OR ("step"."time"[0, 4] <> 0)) THEN
       "hmi".recipeStepQuantity := 4;
   END_IF;
   IF ("hmi".recipeStepQuantity < 4) AND (("inputs".inputSequence[0, 3] <> 0) OR ("inputs".maskSequence[0, 3] <> 0) OR ("outputs".outputSequence[0, 3] <> 0) OR ("outputs".maskSequence[0, 3] <> 0) OR ("step"."time"[0, 3] <> 0)) THEN
       "hmi".recipeStepQuantity := 3;
   END_IF;
   IF ("hmi".recipeStepQuantity < 3) AND (("inputs".inputSequence[0, 2] <> 0) OR ("inputs".maskSequence[0, 2] <> 0) OR ("outputs".outputSequence[0, 2] <> 0) OR ("outputs".maskSequence[0, 2] <> 0) OR ("step"."time"[0, 2] <> 0)) THEN
       "hmi".recipeStepQuantity := 2;
   END_IF;
   IF ("hmi".recipeStepQuantity < 2) AND (("inputs".inputSequence[0, 1] <> 0) OR ("inputs".maskSequence[0, 1] <> 0) OR ("outputs".outputSequence[0, 1] <> 0) OR ("outputs".maskSequence[0, 1] <> 0) OR ("step"."time"[0, 1] <> 0)) THEN
       "hmi".recipeStepQuantity := 1;
   END_IF;
   IF "hmi".recipeStepQuantity < 1 THEN "hmi".recipeStepQuantity := 0; END_IF;
   IF ("inputs".inputSequence[0, "hmi".recipeStepQuantity] = 0) AND ("inputs".maskSequence[0, "hmi".recipeStepQuantity] = 0) AND ("outputs".outputSequence[0, "hmi".recipeStepQuantity] = 0) AND ("outputs".maskSequence[0, "hmi".recipeStepQuantity] = 0) AND ("step"."time"[0, "hmi".recipeStepQuantity] = 0) AND ("hmi".recipeStepQuantity <> 0) THEN
       "hmi".recipeStepQuantity := "hmi".recipeStepQuantity - 1;
   END_IF;
END_REGION

REGION Network 9: INPUTS STATUS TO SHOW ON SCREEN
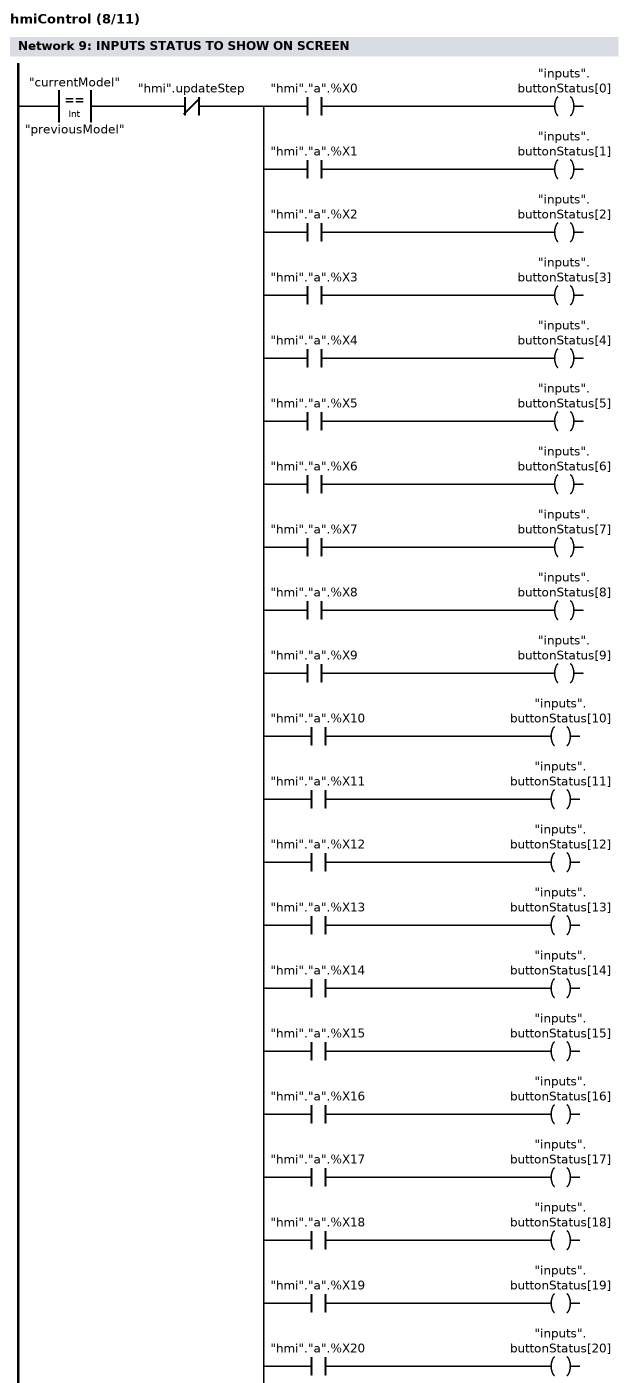
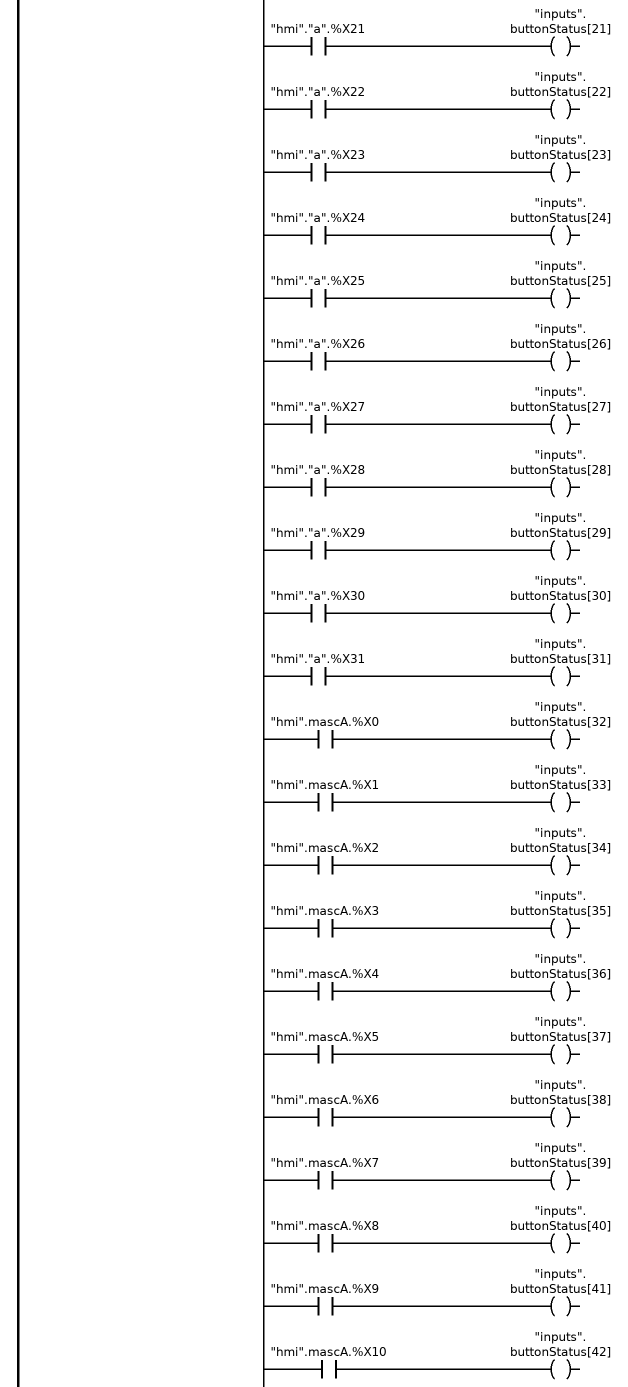
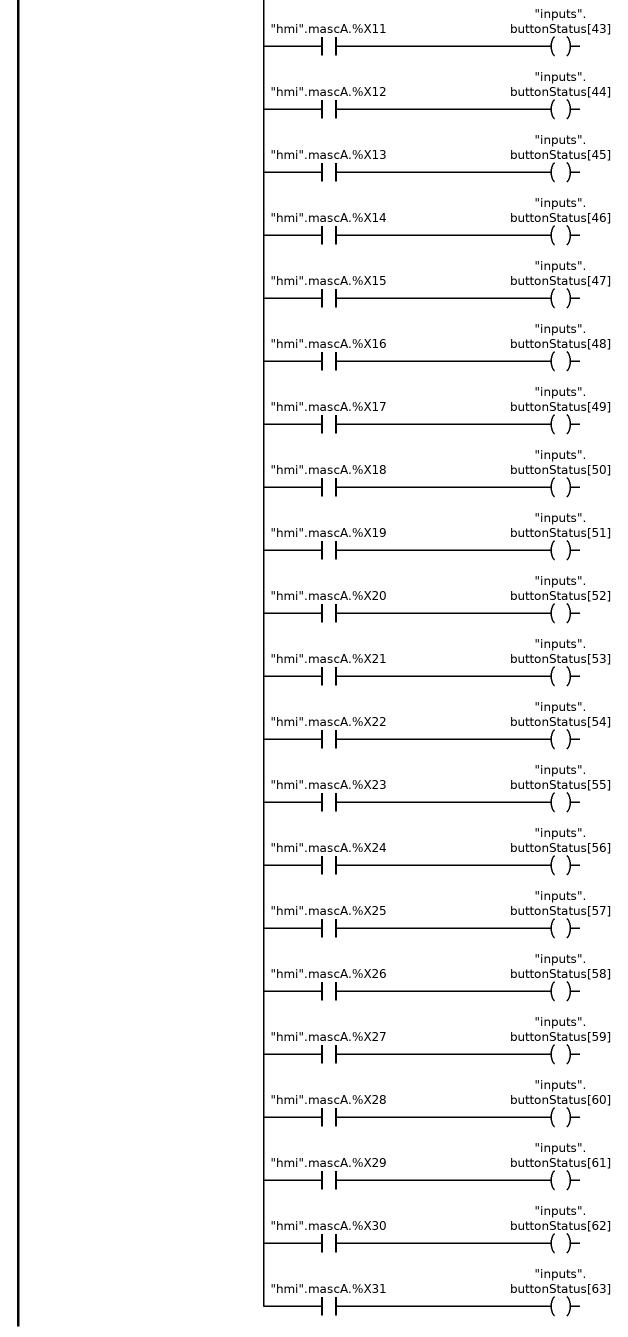
   RUNG wire#powerrail
      { S7_Templates := "SrcType := Int" } EQ_Contact(in1 := "currentModel", in2 := "previousModel")
      I_Contact( "hmi".updateStep )
      wire#w1
      Contact( "hmi"."a".%X0 )
      Coil( "inputs".buttonStatus[0] )
   END_RUNG
   RUNG wire#w1
      Contact( "hmi"."a".%X1 )
      Coil( "inputs".buttonStatus[1] )
   END_RUNG
   RUNG wire#w1
      Contact( "hmi"."a".%X2 )
      Coil( "inputs".buttonStatus[2] )
   END_RUNG
   RUNG wire#w1
      Contact( "hmi"."a".%X3 )
      Coil( "inputs".buttonStatus[3] )
   END_RUNG
   RUNG wire#w1
      Contact( "hmi"."a".%X4 )
      Coil( "inputs".buttonStatus[4] )
   END_RUNG
   RUNG wire#w1
      Contact( "hmi"."a".%X5 )
      Coil( "inputs".buttonStatus[5] )
   END_RUNG
   RUNG wire#w1
      Contact( "hmi"."a".%X6 )
      Coil( "inputs".buttonStatus[6] )
   END_RUNG
   RUNG wire#w1
      Contact( "hmi"."a".%X7 )
      Coil( "inputs".buttonStatus[7] )
   END_RUNG
   RUNG wire#w1
      Contact( "hmi"."a".%X8 )
      Coil( "inputs".buttonStatus[8] )
   END_RUNG
   RUNG wire#w1
      Contact( "hmi"."a".%X9 )
      Coil( "inputs".buttonStatus[9] )
   END_RUNG
   RUNG wire#w1
      Contact( "hmi"."a".%X10 )
      Coil( "inputs".buttonStatus[10] )
   END_RUNG
   RUNG wire#w1
      Contact( "hmi"."a".%X11 )
      Coil( "inputs".buttonStatus[11] )
   END_RUNG
   RUNG wire#w1
      Contact( "hmi"."a".%X12 )
      Coil( "inputs".buttonStatus[12] )
   END_RUNG
   RUNG wire#w1
      Contact( "hmi"."a".%X13 )
      Coil( "inputs".buttonStatus[13] )
   END_RUNG
   RUNG wire#w1
      Contact( "hmi"."a".%X14 )
      Coil( "inputs".buttonStatus[14] )
   END_RUNG
   RUNG wire#w1
      Contact( "hmi"."a".%X15 )
      Coil( "inputs".buttonStatus[15] )
   END_RUNG
   RUNG wire#w1
      Contact( "hmi"."a".%X16 )
      Coil( "inputs".buttonStatus[16] )
   END_RUNG
   RUNG wire#w1
      Contact( "hmi"."a".%X17 )
      Coil( "inputs".buttonStatus[17] )
   END_RUNG
   RUNG wire#w1
      Contact( "hmi"."a".%X18 )
      Coil( "inputs".buttonStatus[18] )
   END_RUNG
   RUNG wire#w1
      Contact( "hmi"."a".%X19 )
      Coil( "inputs".buttonStatus[19] )
   END_RUNG
   RUNG wire#w1
      Contact( "hmi"."a".%X20 )
      Coil( "inputs".buttonStatus[20] )
   END_RUNG
   RUNG wire#w1
      Contact( "hmi"."a".%X21 )
      Coil( "inputs".buttonStatus[21] )
   END_RUNG
   RUNG wire#w1
      Contact( "hmi"."a".%X22 )
      Coil( "inputs".buttonStatus[22] )
   END_RUNG
   RUNG wire#w1
      Contact( "hmi"."a".%X23 )
      Coil( "inputs".buttonStatus[23] )
   END_RUNG
   RUNG wire#w1
      Contact( "hmi"."a".%X24 )
      Coil( "inputs".buttonStatus[24] )
   END_RUNG
   RUNG wire#w1
      Contact( "hmi"."a".%X25 )
      Coil( "inputs".buttonStatus[25] )
   END_RUNG
   RUNG wire#w1
      Contact( "hmi"."a".%X26 )
      Coil( "inputs".buttonStatus[26] )
   END_RUNG
   RUNG wire#w1
      Contact( "hmi"."a".%X27 )
      Coil( "inputs".buttonStatus[27] )
   END_RUNG
   RUNG wire#w1
      Contact( "hmi"."a".%X28 )
      Coil( "inputs".buttonStatus[28] )
   END_RUNG
   RUNG wire#w1
      Contact( "hmi"."a".%X29 )
      Coil( "inputs".buttonStatus[29] )
   END_RUNG
   RUNG wire#w1
      Contact( "hmi"."a".%X30 )
      Coil( "inputs".buttonStatus[30] )
   END_RUNG
   RUNG wire#w1
      Contact( "hmi"."a".%X31 )
      Coil( "inputs".buttonStatus[31] )
   END_RUNG
   RUNG wire#w1
      Contact( "hmi".mascA.%X0 )
      Coil( "inputs".buttonStatus[32] )
   END_RUNG
   RUNG wire#w1
      Contact( "hmi".mascA.%X1 )
      Coil( "inputs".buttonStatus[33] )
   END_RUNG
   RUNG wire#w1
      Contact( "hmi".mascA.%X2 )
      Coil( "inputs".buttonStatus[34] )
   END_RUNG
   RUNG wire#w1
      Contact( "hmi".mascA.%X3 )
      Coil( "inputs".buttonStatus[35] )
   END_RUNG
   RUNG wire#w1
      Contact( "hmi".mascA.%X4 )
      Coil( "inputs".buttonStatus[36] )
   END_RUNG
   RUNG wire#w1
      Contact( "hmi".mascA.%X5 )
      Coil( "inputs".buttonStatus[37] )
   END_RUNG
   RUNG wire#w1
      Contact( "hmi".mascA.%X6 )
      Coil( "inputs".buttonStatus[38] )
   END_RUNG
   RUNG wire#w1
      Contact( "hmi".mascA.%X7 )
      Coil( "inputs".buttonStatus[39] )
   END_RUNG
   RUNG wire#w1
      Contact( "hmi".mascA.%X8 )
      Coil( "inputs".buttonStatus[40] )
   END_RUNG
   RUNG wire#w1
      Contact( "hmi".mascA.%X9 )
      Coil( "inputs".buttonStatus[41] )
   END_RUNG
   RUNG wire#w1
      Contact( "hmi".mascA.%X10 )
      Coil( "inputs".buttonStatus[42] )
   END_RUNG
   RUNG wire#w1
      Contact( "hmi".mascA.%X11 )
      Coil( "inputs".buttonStatus[43] )
   END_RUNG
   RUNG wire#w1
      Contact( "hmi".mascA.%X12 )
      Coil( "inputs".buttonStatus[44] )
   END_RUNG
   RUNG wire#w1
      Contact( "hmi".mascA.%X13 )
      Coil( "inputs".buttonStatus[45] )
   END_RUNG
   RUNG wire#w1
      Contact( "hmi".mascA.%X14 )
      Coil( "inputs".buttonStatus[46] )
   END_RUNG
   RUNG wire#w1
      Contact( "hmi".mascA.%X15 )
      Coil( "inputs".buttonStatus[47] )
   END_RUNG
   RUNG wire#w1
      Contact( "hmi".mascA.%X16 )
      Coil( "inputs".buttonStatus[48] )
   END_RUNG
   RUNG wire#w1
      Contact( "hmi".mascA.%X17 )
      Coil( "inputs".buttonStatus[49] )
   END_RUNG
   RUNG wire#w1
      Contact( "hmi".mascA.%X18 )
      Coil( "inputs".buttonStatus[50] )
   END_RUNG
   RUNG wire#w1
      Contact( "hmi".mascA.%X19 )
      Coil( "inputs".buttonStatus[51] )
   END_RUNG
   RUNG wire#w1
      Contact( "hmi".mascA.%X20 )
      Coil( "inputs".buttonStatus[52] )
   END_RUNG
   RUNG wire#w1
      Contact( "hmi".mascA.%X21 )
      Coil( "inputs".buttonStatus[53] )
   END_RUNG
   RUNG wire#w1
      Contact( "hmi".mascA.%X22 )
      Coil( "inputs".buttonStatus[54] )
   END_RUNG
   RUNG wire#w1
      Contact( "hmi".mascA.%X23 )
      Coil( "inputs".buttonStatus[55] )
   END_RUNG
   RUNG wire#w1
      Contact( "hmi".mascA.%X24 )
      Coil( "inputs".buttonStatus[56] )
   END_RUNG
   RUNG wire#w1
      Contact( "hmi".mascA.%X25 )
      Coil( "inputs".buttonStatus[57] )
   END_RUNG
   RUNG wire#w1
      Contact( "hmi".mascA.%X26 )
      Coil( "inputs".buttonStatus[58] )
   END_RUNG
   RUNG wire#w1
      Contact( "hmi".mascA.%X27 )
      Coil( "inputs".buttonStatus[59] )
   END_RUNG
   RUNG wire#w1
      Contact( "hmi".mascA.%X28 )
      Coil( "inputs".buttonStatus[60] )
   END_RUNG
   RUNG wire#w1
      Contact( "hmi".mascA.%X29 )
      Coil( "inputs".buttonStatus[61] )
   END_RUNG
   RUNG wire#w1
      Contact( "hmi".mascA.%X30 )
      Coil( "inputs".buttonStatus[62] )
   END_RUNG
   RUNG wire#w1
      Contact( "hmi".mascA.%X31 )
      Coil( "inputs".buttonStatus[63] )
   END_RUNG
   // the same network as SCL:
   #_w1 := ("currentModel" = "previousModel") AND NOT "hmi".updateStep;
   "inputs".buttonStatus[0] := #_w1 AND "hmi"."a".%X0;
   "inputs".buttonStatus[1] := #_w1 AND "hmi"."a".%X1;
   "inputs".buttonStatus[2] := #_w1 AND "hmi"."a".%X2;
   "inputs".buttonStatus[3] := #_w1 AND "hmi"."a".%X3;
   "inputs".buttonStatus[4] := #_w1 AND "hmi"."a".%X4;
   "inputs".buttonStatus[5] := #_w1 AND "hmi"."a".%X5;
   "inputs".buttonStatus[6] := #_w1 AND "hmi"."a".%X6;
   "inputs".buttonStatus[7] := #_w1 AND "hmi"."a".%X7;
   "inputs".buttonStatus[8] := #_w1 AND "hmi"."a".%X8;
   "inputs".buttonStatus[9] := #_w1 AND "hmi"."a".%X9;
   "inputs".buttonStatus[10] := #_w1 AND "hmi"."a".%X10;
   "inputs".buttonStatus[11] := #_w1 AND "hmi"."a".%X11;
   "inputs".buttonStatus[12] := #_w1 AND "hmi"."a".%X12;
   "inputs".buttonStatus[13] := #_w1 AND "hmi"."a".%X13;
   "inputs".buttonStatus[14] := #_w1 AND "hmi"."a".%X14;
   "inputs".buttonStatus[15] := #_w1 AND "hmi"."a".%X15;
   "inputs".buttonStatus[16] := #_w1 AND "hmi"."a".%X16;
   "inputs".buttonStatus[17] := #_w1 AND "hmi"."a".%X17;
   "inputs".buttonStatus[18] := #_w1 AND "hmi"."a".%X18;
   "inputs".buttonStatus[19] := #_w1 AND "hmi"."a".%X19;
   "inputs".buttonStatus[20] := #_w1 AND "hmi"."a".%X20;
   "inputs".buttonStatus[21] := #_w1 AND "hmi"."a".%X21;
   "inputs".buttonStatus[22] := #_w1 AND "hmi"."a".%X22;
   "inputs".buttonStatus[23] := #_w1 AND "hmi"."a".%X23;
   "inputs".buttonStatus[24] := #_w1 AND "hmi"."a".%X24;
   "inputs".buttonStatus[25] := #_w1 AND "hmi"."a".%X25;
   "inputs".buttonStatus[26] := #_w1 AND "hmi"."a".%X26;
   "inputs".buttonStatus[27] := #_w1 AND "hmi"."a".%X27;
   "inputs".buttonStatus[28] := #_w1 AND "hmi"."a".%X28;
   "inputs".buttonStatus[29] := #_w1 AND "hmi"."a".%X29;
   "inputs".buttonStatus[30] := #_w1 AND "hmi"."a".%X30;
   "inputs".buttonStatus[31] := #_w1 AND "hmi"."a".%X31;
   "inputs".buttonStatus[32] := #_w1 AND "hmi".mascA.%X0;
   "inputs".buttonStatus[33] := #_w1 AND "hmi".mascA.%X1;
   "inputs".buttonStatus[34] := #_w1 AND "hmi".mascA.%X2;
   "inputs".buttonStatus[35] := #_w1 AND "hmi".mascA.%X3;
   "inputs".buttonStatus[36] := #_w1 AND "hmi".mascA.%X4;
   "inputs".buttonStatus[37] := #_w1 AND "hmi".mascA.%X5;
   "inputs".buttonStatus[38] := #_w1 AND "hmi".mascA.%X6;
   "inputs".buttonStatus[39] := #_w1 AND "hmi".mascA.%X7;
   "inputs".buttonStatus[40] := #_w1 AND "hmi".mascA.%X8;
   "inputs".buttonStatus[41] := #_w1 AND "hmi".mascA.%X9;
   "inputs".buttonStatus[42] := #_w1 AND "hmi".mascA.%X10;
   "inputs".buttonStatus[43] := #_w1 AND "hmi".mascA.%X11;
   "inputs".buttonStatus[44] := #_w1 AND "hmi".mascA.%X12;
   "inputs".buttonStatus[45] := #_w1 AND "hmi".mascA.%X13;
   "inputs".buttonStatus[46] := #_w1 AND "hmi".mascA.%X14;
   "inputs".buttonStatus[47] := #_w1 AND "hmi".mascA.%X15;
   "inputs".buttonStatus[48] := #_w1 AND "hmi".mascA.%X16;
   "inputs".buttonStatus[49] := #_w1 AND "hmi".mascA.%X17;
   "inputs".buttonStatus[50] := #_w1 AND "hmi".mascA.%X18;
   "inputs".buttonStatus[51] := #_w1 AND "hmi".mascA.%X19;
   "inputs".buttonStatus[52] := #_w1 AND "hmi".mascA.%X20;
   "inputs".buttonStatus[53] := #_w1 AND "hmi".mascA.%X21;
   "inputs".buttonStatus[54] := #_w1 AND "hmi".mascA.%X22;
   "inputs".buttonStatus[55] := #_w1 AND "hmi".mascA.%X23;
   "inputs".buttonStatus[56] := #_w1 AND "hmi".mascA.%X24;
   "inputs".buttonStatus[57] := #_w1 AND "hmi".mascA.%X25;
   "inputs".buttonStatus[58] := #_w1 AND "hmi".mascA.%X26;
   "inputs".buttonStatus[59] := #_w1 AND "hmi".mascA.%X27;
   "inputs".buttonStatus[60] := #_w1 AND "hmi".mascA.%X28;
   "inputs".buttonStatus[61] := #_w1 AND "hmi".mascA.%X29;
   "inputs".buttonStatus[62] := #_w1 AND "hmi".mascA.%X30;
   "inputs".buttonStatus[63] := #_w1 AND "hmi".mascA.%X31;
END_REGION

REGION Network 10: OUTPUTS STATUS TO SHOW ON SCREEN
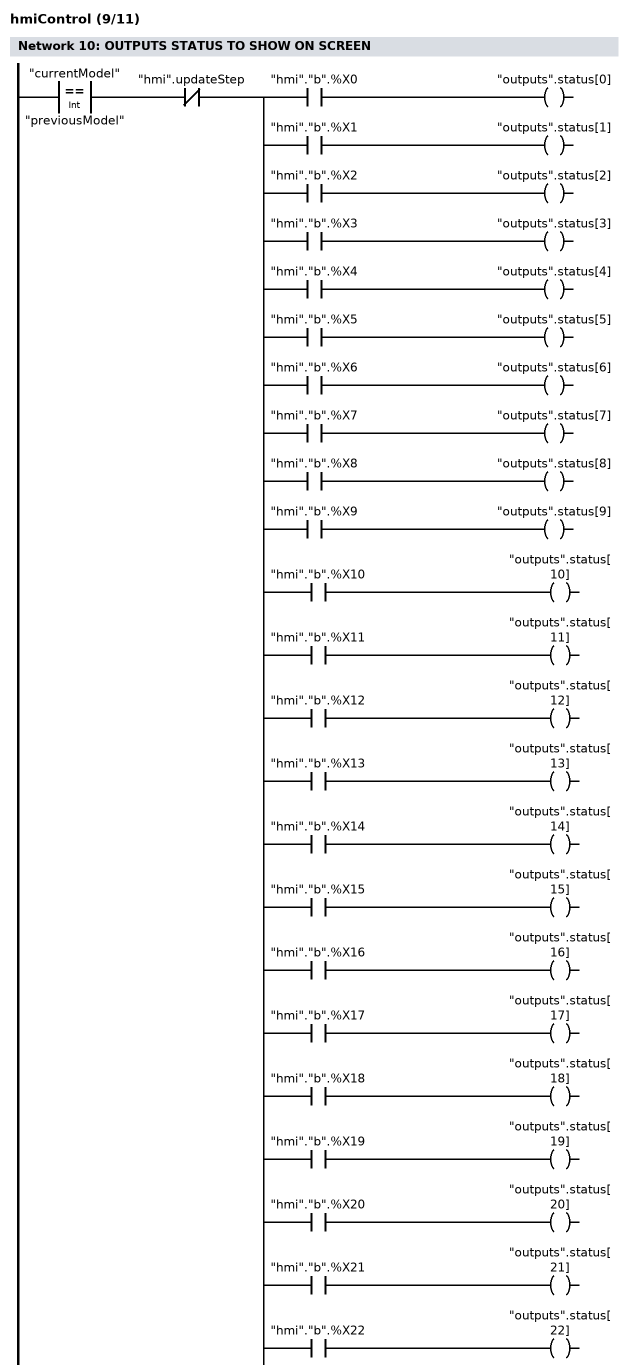
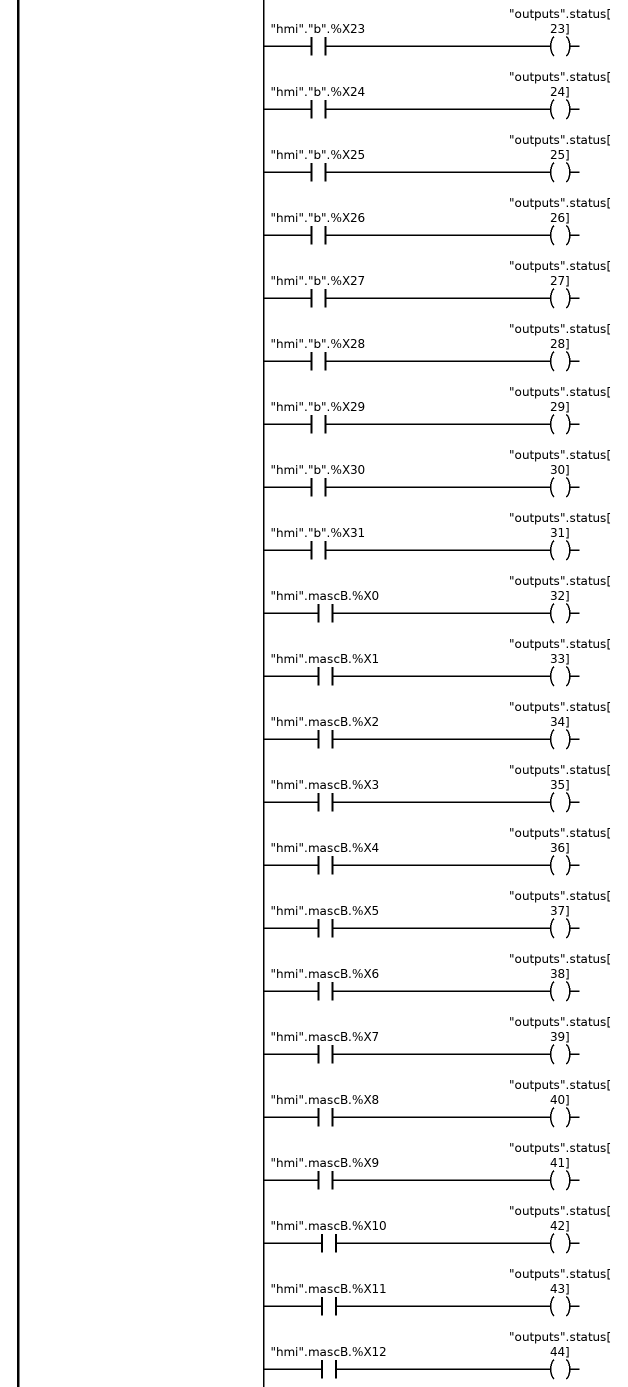
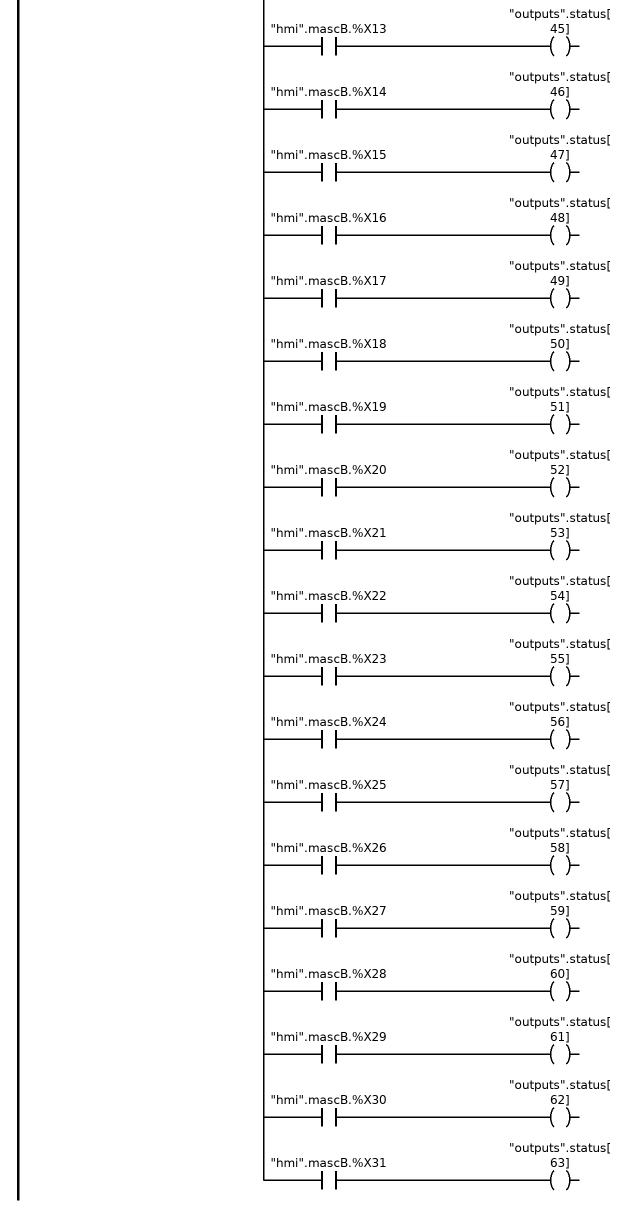
   RUNG wire#powerrail
      { S7_Templates := "SrcType := Int" } EQ_Contact(in1 := "currentModel", in2 := "previousModel")
      I_Contact( "hmi".updateStep )
      wire#w1
      Contact( "hmi"."b".%X0 )
      Coil( "outputs".status[0] )
   END_RUNG
   RUNG wire#w1
      Contact( "hmi"."b".%X1 )
      Coil( "outputs".status[1] )
   END_RUNG
   RUNG wire#w1
      Contact( "hmi"."b".%X2 )
      Coil( "outputs".status[2] )
   END_RUNG
   RUNG wire#w1
      Contact( "hmi"."b".%X3 )
      Coil( "outputs".status[3] )
   END_RUNG
   RUNG wire#w1
      Contact( "hmi"."b".%X4 )
      Coil( "outputs".status[4] )
   END_RUNG
   RUNG wire#w1
      Contact( "hmi"."b".%X5 )
      Coil( "outputs".status[5] )
   END_RUNG
   RUNG wire#w1
      Contact( "hmi"."b".%X6 )
      Coil( "outputs".status[6] )
   END_RUNG
   RUNG wire#w1
      Contact( "hmi"."b".%X7 )
      Coil( "outputs".status[7] )
   END_RUNG
   RUNG wire#w1
      Contact( "hmi"."b".%X8 )
      Coil( "outputs".status[8] )
   END_RUNG
   RUNG wire#w1
      Contact( "hmi"."b".%X9 )
      Coil( "outputs".status[9] )
   END_RUNG
   RUNG wire#w1
      Contact( "hmi"."b".%X10 )
      Coil( "outputs".status[10] )
   END_RUNG
   RUNG wire#w1
      Contact( "hmi"."b".%X11 )
      Coil( "outputs".status[11] )
   END_RUNG
   RUNG wire#w1
      Contact( "hmi"."b".%X12 )
      Coil( "outputs".status[12] )
   END_RUNG
   RUNG wire#w1
      Contact( "hmi"."b".%X13 )
      Coil( "outputs".status[13] )
   END_RUNG
   RUNG wire#w1
      Contact( "hmi"."b".%X14 )
      Coil( "outputs".status[14] )
   END_RUNG
   RUNG wire#w1
      Contact( "hmi"."b".%X15 )
      Coil( "outputs".status[15] )
   END_RUNG
   RUNG wire#w1
      Contact( "hmi"."b".%X16 )
      Coil( "outputs".status[16] )
   END_RUNG
   RUNG wire#w1
      Contact( "hmi"."b".%X17 )
      Coil( "outputs".status[17] )
   END_RUNG
   RUNG wire#w1
      Contact( "hmi"."b".%X18 )
      Coil( "outputs".status[18] )
   END_RUNG
   RUNG wire#w1
      Contact( "hmi"."b".%X19 )
      Coil( "outputs".status[19] )
   END_RUNG
   RUNG wire#w1
      Contact( "hmi"."b".%X20 )
      Coil( "outputs".status[20] )
   END_RUNG
   RUNG wire#w1
      Contact( "hmi"."b".%X21 )
      Coil( "outputs".status[21] )
   END_RUNG
   RUNG wire#w1
      Contact( "hmi"."b".%X22 )
      Coil( "outputs".status[22] )
   END_RUNG
   RUNG wire#w1
      Contact( "hmi"."b".%X23 )
      Coil( "outputs".status[23] )
   END_RUNG
   RUNG wire#w1
      Contact( "hmi"."b".%X24 )
      Coil( "outputs".status[24] )
   END_RUNG
   RUNG wire#w1
      Contact( "hmi"."b".%X25 )
      Coil( "outputs".status[25] )
   END_RUNG
   RUNG wire#w1
      Contact( "hmi"."b".%X26 )
      Coil( "outputs".status[26] )
   END_RUNG
   RUNG wire#w1
      Contact( "hmi"."b".%X27 )
      Coil( "outputs".status[27] )
   END_RUNG
   RUNG wire#w1
      Contact( "hmi"."b".%X28 )
      Coil( "outputs".status[28] )
   END_RUNG
   RUNG wire#w1
      Contact( "hmi"."b".%X29 )
      Coil( "outputs".status[29] )
   END_RUNG
   RUNG wire#w1
      Contact( "hmi"."b".%X30 )
      Coil( "outputs".status[30] )
   END_RUNG
   RUNG wire#w1
      Contact( "hmi"."b".%X31 )
      Coil( "outputs".status[31] )
   END_RUNG
   RUNG wire#w1
      Contact( "hmi".mascB.%X0 )
      Coil( "outputs".status[32] )
   END_RUNG
   RUNG wire#w1
      Contact( "hmi".mascB.%X1 )
      Coil( "outputs".status[33] )
   END_RUNG
   RUNG wire#w1
      Contact( "hmi".mascB.%X2 )
      Coil( "outputs".status[34] )
   END_RUNG
   RUNG wire#w1
      Contact( "hmi".mascB.%X3 )
      Coil( "outputs".status[35] )
   END_RUNG
   RUNG wire#w1
      Contact( "hmi".mascB.%X4 )
      Coil( "outputs".status[36] )
   END_RUNG
   RUNG wire#w1
      Contact( "hmi".mascB.%X5 )
      Coil( "outputs".status[37] )
   END_RUNG
   RUNG wire#w1
      Contact( "hmi".mascB.%X6 )
      Coil( "outputs".status[38] )
   END_RUNG
   RUNG wire#w1
      Contact( "hmi".mascB.%X7 )
      Coil( "outputs".status[39] )
   END_RUNG
   RUNG wire#w1
      Contact( "hmi".mascB.%X8 )
      Coil( "outputs".status[40] )
   END_RUNG
   RUNG wire#w1
      Contact( "hmi".mascB.%X9 )
      Coil( "outputs".status[41] )
   END_RUNG
   RUNG wire#w1
      Contact( "hmi".mascB.%X10 )
      Coil( "outputs".status[42] )
   END_RUNG
   RUNG wire#w1
      Contact( "hmi".mascB.%X11 )
      Coil( "outputs".status[43] )
   END_RUNG
   RUNG wire#w1
      Contact( "hmi".mascB.%X12 )
      Coil( "outputs".status[44] )
   END_RUNG
   RUNG wire#w1
      Contact( "hmi".mascB.%X13 )
      Coil( "outputs".status[45] )
   END_RUNG
   RUNG wire#w1
      Contact( "hmi".mascB.%X14 )
      Coil( "outputs".status[46] )
   END_RUNG
   RUNG wire#w1
      Contact( "hmi".mascB.%X15 )
      Coil( "outputs".status[47] )
   END_RUNG
   RUNG wire#w1
      Contact( "hmi".mascB.%X16 )
      Coil( "outputs".status[48] )
   END_RUNG
   RUNG wire#w1
      Contact( "hmi".mascB.%X17 )
      Coil( "outputs".status[49] )
   END_RUNG
   RUNG wire#w1
      Contact( "hmi".mascB.%X18 )
      Coil( "outputs".status[50] )
   END_RUNG
   RUNG wire#w1
      Contact( "hmi".mascB.%X19 )
      Coil( "outputs".status[51] )
   END_RUNG
   RUNG wire#w1
      Contact( "hmi".mascB.%X20 )
      Coil( "outputs".status[52] )
   END_RUNG
   RUNG wire#w1
      Contact( "hmi".mascB.%X21 )
      Coil( "outputs".status[53] )
   END_RUNG
   RUNG wire#w1
      Contact( "hmi".mascB.%X22 )
      Coil( "outputs".status[54] )
   END_RUNG
   RUNG wire#w1
      Contact( "hmi".mascB.%X23 )
      Coil( "outputs".status[55] )
   END_RUNG
   RUNG wire#w1
      Contact( "hmi".mascB.%X24 )
      Coil( "outputs".status[56] )
   END_RUNG
   RUNG wire#w1
      Contact( "hmi".mascB.%X25 )
      Coil( "outputs".status[57] )
   END_RUNG
   RUNG wire#w1
      Contact( "hmi".mascB.%X26 )
      Coil( "outputs".status[58] )
   END_RUNG
   RUNG wire#w1
      Contact( "hmi".mascB.%X27 )
      Coil( "outputs".status[59] )
   END_RUNG
   RUNG wire#w1
      Contact( "hmi".mascB.%X28 )
      Coil( "outputs".status[60] )
   END_RUNG
   RUNG wire#w1
      Contact( "hmi".mascB.%X29 )
      Coil( "outputs".status[61] )
   END_RUNG
   RUNG wire#w1
      Contact( "hmi".mascB.%X30 )
      Coil( "outputs".status[62] )
   END_RUNG
   RUNG wire#w1
      Contact( "hmi".mascB.%X31 )
      Coil( "outputs".status[63] )
   END_RUNG
   // the same network as SCL:
   #_w1 := ("currentModel" = "previousModel") AND NOT "hmi".updateStep;
   "outputs".status[0] := #_w1 AND "hmi"."b".%X0;
   "outputs".status[1] := #_w1 AND "hmi"."b".%X1;
   "outputs".status[2] := #_w1 AND "hmi"."b".%X2;
   "outputs".status[3] := #_w1 AND "hmi"."b".%X3;
   "outputs".status[4] := #_w1 AND "hmi"."b".%X4;
   "outputs".status[5] := #_w1 AND "hmi"."b".%X5;
   "outputs".status[6] := #_w1 AND "hmi"."b".%X6;
   "outputs".status[7] := #_w1 AND "hmi"."b".%X7;
   "outputs".status[8] := #_w1 AND "hmi"."b".%X8;
   "outputs".status[9] := #_w1 AND "hmi"."b".%X9;
   "outputs".status[10] := #_w1 AND "hmi"."b".%X10;
   "outputs".status[11] := #_w1 AND "hmi"."b".%X11;
   "outputs".status[12] := #_w1 AND "hmi"."b".%X12;
   "outputs".status[13] := #_w1 AND "hmi"."b".%X13;
   "outputs".status[14] := #_w1 AND "hmi"."b".%X14;
   "outputs".status[15] := #_w1 AND "hmi"."b".%X15;
   "outputs".status[16] := #_w1 AND "hmi"."b".%X16;
   "outputs".status[17] := #_w1 AND "hmi"."b".%X17;
   "outputs".status[18] := #_w1 AND "hmi"."b".%X18;
   "outputs".status[19] := #_w1 AND "hmi"."b".%X19;
   "outputs".status[20] := #_w1 AND "hmi"."b".%X20;
   "outputs".status[21] := #_w1 AND "hmi"."b".%X21;
   "outputs".status[22] := #_w1 AND "hmi"."b".%X22;
   "outputs".status[23] := #_w1 AND "hmi"."b".%X23;
   "outputs".status[24] := #_w1 AND "hmi"."b".%X24;
   "outputs".status[25] := #_w1 AND "hmi"."b".%X25;
   "outputs".status[26] := #_w1 AND "hmi"."b".%X26;
   "outputs".status[27] := #_w1 AND "hmi"."b".%X27;
   "outputs".status[28] := #_w1 AND "hmi"."b".%X28;
   "outputs".status[29] := #_w1 AND "hmi"."b".%X29;
   "outputs".status[30] := #_w1 AND "hmi"."b".%X30;
   "outputs".status[31] := #_w1 AND "hmi"."b".%X31;
   "outputs".status[32] := #_w1 AND "hmi".mascB.%X0;
   "outputs".status[33] := #_w1 AND "hmi".mascB.%X1;
   "outputs".status[34] := #_w1 AND "hmi".mascB.%X2;
   "outputs".status[35] := #_w1 AND "hmi".mascB.%X3;
   "outputs".status[36] := #_w1 AND "hmi".mascB.%X4;
   "outputs".status[37] := #_w1 AND "hmi".mascB.%X5;
   "outputs".status[38] := #_w1 AND "hmi".mascB.%X6;
   "outputs".status[39] := #_w1 AND "hmi".mascB.%X7;
   "outputs".status[40] := #_w1 AND "hmi".mascB.%X8;
   "outputs".status[41] := #_w1 AND "hmi".mascB.%X9;
   "outputs".status[42] := #_w1 AND "hmi".mascB.%X10;
   "outputs".status[43] := #_w1 AND "hmi".mascB.%X11;
   "outputs".status[44] := #_w1 AND "hmi".mascB.%X12;
   "outputs".status[45] := #_w1 AND "hmi".mascB.%X13;
   "outputs".status[46] := #_w1 AND "hmi".mascB.%X14;
   "outputs".status[47] := #_w1 AND "hmi".mascB.%X15;
   "outputs".status[48] := #_w1 AND "hmi".mascB.%X16;
   "outputs".status[49] := #_w1 AND "hmi".mascB.%X17;
   "outputs".status[50] := #_w1 AND "hmi".mascB.%X18;
   "outputs".status[51] := #_w1 AND "hmi".mascB.%X19;
   "outputs".status[52] := #_w1 AND "hmi".mascB.%X20;
   "outputs".status[53] := #_w1 AND "hmi".mascB.%X21;
   "outputs".status[54] := #_w1 AND "hmi".mascB.%X22;
   "outputs".status[55] := #_w1 AND "hmi".mascB.%X23;
   "outputs".status[56] := #_w1 AND "hmi".mascB.%X24;
   "outputs".status[57] := #_w1 AND "hmi".mascB.%X25;
   "outputs".status[58] := #_w1 AND "hmi".mascB.%X26;
   "outputs".status[59] := #_w1 AND "hmi".mascB.%X27;
   "outputs".status[60] := #_w1 AND "hmi".mascB.%X28;
   "outputs".status[61] := #_w1 AND "hmi".mascB.%X29;
   "outputs".status[62] := #_w1 AND "hmi".mascB.%X30;
   "outputs".status[63] := #_w1 AND "hmi".mascB.%X31;
END_REGION

REGION Network 11: HOME BUTTON
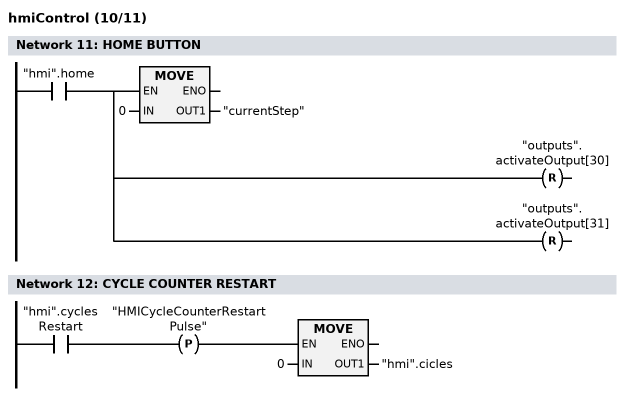
   RUNG wire#powerrail
      Contact( "hmi".home )
      wire#w1
      Move(in := 0, out1 => "currentStep")
   END_RUNG
   RUNG wire#w1
      R_Coil( "outputs".activateOutput[30] )
   END_RUNG
   RUNG wire#w1
      R_Coil( "outputs".activateOutput[31] )
   END_RUNG
   // the same network as SCL:
   IF "hmi".home THEN
       "currentStep" := 0;
       "outputs".activateOutput[30] := FALSE;
       "outputs".activateOutput[31] := FALSE;
   END_IF;
END_REGION

REGION Network 12: CYCLE COUNTER RESTART
   RUNG wire#powerrail
      Contact( "hmi".cyclesRestart )
      P_Trig( "HMICycleCounterRestartPulse" )
      Move(in := 0, out1 => "hmi".cicles)
   END_RUNG
   // the same network as SCL:
   #_w1 := "hmi".cyclesRestart AND NOT "HMICycleCounterRestartPulse";   // rising edge
   "HMICycleCounterRestartPulse" := "hmi".cyclesRestart;
   IF #_w1 THEN "hmi".cicles := 0; END_IF;
END_REGION

REGION Network 13: MODEL SELECTION
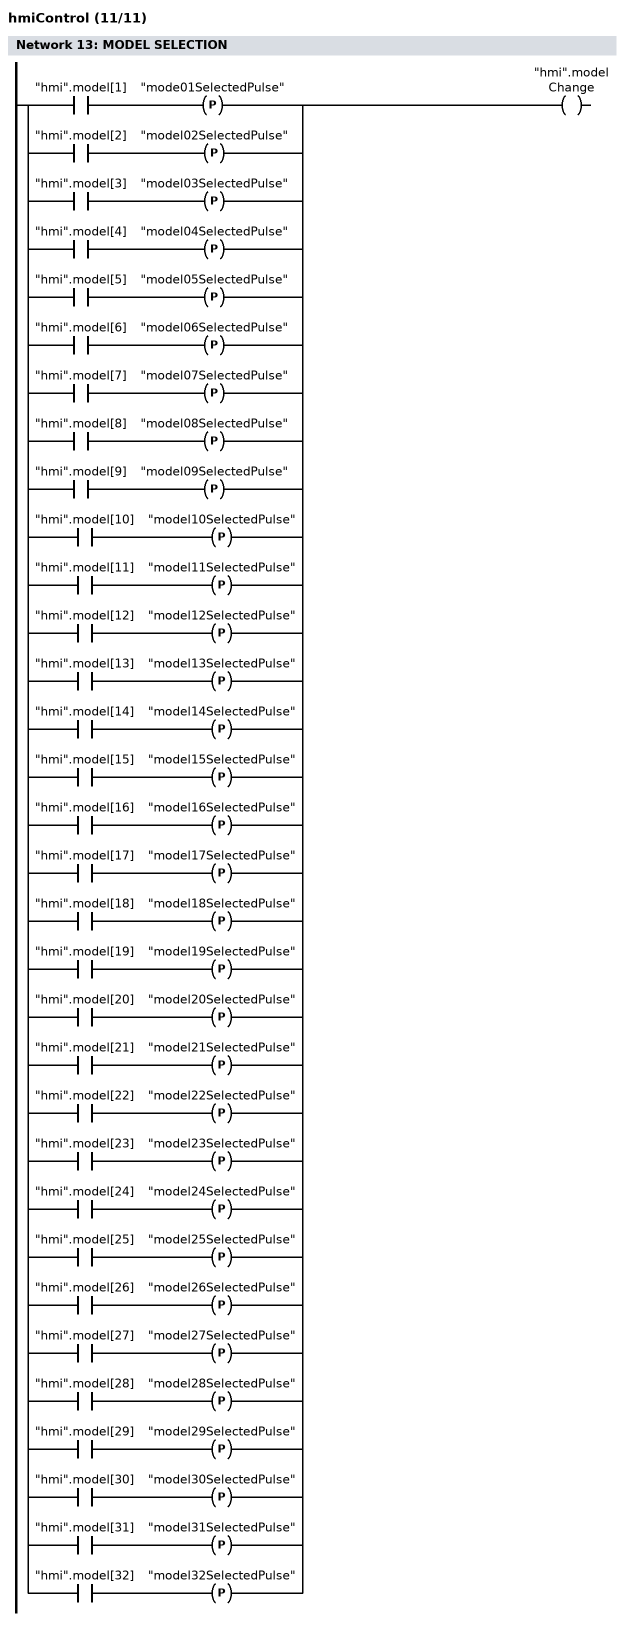
   RUNG wire#powerrail
      Contact( "hmi".model[1] )
      P_Trig( "mode01SelectedPulse" )
      wire#w1
      Coil( "hmi".modelChange )
   END_RUNG
   RUNG wire#powerrail
      Contact( "hmi".model[2] )
      P_Trig( "model02SelectedPulse" )
   END_RUNG wire#w1
   RUNG wire#powerrail
      Contact( "hmi".model[3] )
      P_Trig( "model03SelectedPulse" )
   END_RUNG wire#w1
   RUNG wire#powerrail
      Contact( "hmi".model[4] )
      P_Trig( "model04SelectedPulse" )
   END_RUNG wire#w1
   RUNG wire#powerrail
      Contact( "hmi".model[5] )
      P_Trig( "model05SelectedPulse" )
   END_RUNG wire#w1
   RUNG wire#powerrail
      Contact( "hmi".model[6] )
      P_Trig( "model06SelectedPulse" )
   END_RUNG wire#w1
   RUNG wire#powerrail
      Contact( "hmi".model[7] )
      P_Trig( "model07SelectedPulse" )
   END_RUNG wire#w1
   RUNG wire#powerrail
      Contact( "hmi".model[8] )
      P_Trig( "model08SelectedPulse" )
   END_RUNG wire#w1
   RUNG wire#powerrail
      Contact( "hmi".model[9] )
      P_Trig( "model09SelectedPulse" )
   END_RUNG wire#w1
   RUNG wire#powerrail
      Contact( "hmi".model[10] )
      P_Trig( "model10SelectedPulse" )
   END_RUNG wire#w1
   RUNG wire#powerrail
      Contact( "hmi".model[11] )
      P_Trig( "model11SelectedPulse" )
   END_RUNG wire#w1
   RUNG wire#powerrail
      Contact( "hmi".model[12] )
      P_Trig( "model12SelectedPulse" )
   END_RUNG wire#w1
   RUNG wire#powerrail
      Contact( "hmi".model[13] )
      P_Trig( "model13SelectedPulse" )
   END_RUNG wire#w1
   RUNG wire#powerrail
      Contact( "hmi".model[14] )
      P_Trig( "model14SelectedPulse" )
   END_RUNG wire#w1
   RUNG wire#powerrail
      Contact( "hmi".model[15] )
      P_Trig( "model15SelectedPulse" )
   END_RUNG wire#w1
   RUNG wire#powerrail
      Contact( "hmi".model[16] )
      P_Trig( "model16SelectedPulse" )
   END_RUNG wire#w1
   RUNG wire#powerrail
      Contact( "hmi".model[17] )
      P_Trig( "model17SelectedPulse" )
   END_RUNG wire#w1
   RUNG wire#powerrail
      Contact( "hmi".model[18] )
      P_Trig( "model18SelectedPulse" )
   END_RUNG wire#w1
   RUNG wire#powerrail
      Contact( "hmi".model[19] )
      P_Trig( "model19SelectedPulse" )
   END_RUNG wire#w1
   RUNG wire#powerrail
      Contact( "hmi".model[20] )
      P_Trig( "model20SelectedPulse" )
   END_RUNG wire#w1
   RUNG wire#powerrail
      Contact( "hmi".model[21] )
      P_Trig( "model21SelectedPulse" )
   END_RUNG wire#w1
   RUNG wire#powerrail
      Contact( "hmi".model[22] )
      P_Trig( "model22SelectedPulse" )
   END_RUNG wire#w1
   RUNG wire#powerrail
      Contact( "hmi".model[23] )
      P_Trig( "model23SelectedPulse" )
   END_RUNG wire#w1
   RUNG wire#powerrail
      Contact( "hmi".model[24] )
      P_Trig( "model24SelectedPulse" )
   END_RUNG wire#w1
   RUNG wire#powerrail
      Contact( "hmi".model[25] )
      P_Trig( "model25SelectedPulse" )
   END_RUNG wire#w1
   RUNG wire#powerrail
      Contact( "hmi".model[26] )
      P_Trig( "model26SelectedPulse" )
   END_RUNG wire#w1
   RUNG wire#powerrail
      Contact( "hmi".model[27] )
      P_Trig( "model27SelectedPulse" )
   END_RUNG wire#w1
   RUNG wire#powerrail
      Contact( "hmi".model[28] )
      P_Trig( "model28SelectedPulse" )
   END_RUNG wire#w1
   RUNG wire#powerrail
      Contact( "hmi".model[29] )
      P_Trig( "model29SelectedPulse" )
   END_RUNG wire#w1
   RUNG wire#powerrail
      Contact( "hmi".model[30] )
      P_Trig( "model30SelectedPulse" )
   END_RUNG wire#w1
   RUNG wire#powerrail
      Contact( "hmi".model[31] )
      P_Trig( "model31SelectedPulse" )
   END_RUNG wire#w1
   RUNG wire#powerrail
      Contact( "hmi".model[32] )
      P_Trig( "model32SelectedPulse" )
   END_RUNG wire#w1
   // the same network as SCL:
   #_w1 := "hmi".model[1] AND NOT "mode01SelectedPulse";   // rising edge
   "mode01SelectedPulse" := "hmi".model[1];
   #_w2 := "hmi".model[2] AND NOT "model02SelectedPulse";   // rising edge
   "model02SelectedPulse" := "hmi".model[2];
   #_w3 := "hmi".model[3] AND NOT "model03SelectedPulse";   // rising edge
   "model03SelectedPulse" := "hmi".model[3];
   #_w4 := "hmi".model[4] AND NOT "model04SelectedPulse";   // rising edge
   "model04SelectedPulse" := "hmi".model[4];
   #_w5 := "hmi".model[5] AND NOT "model05SelectedPulse";   // rising edge
   "model05SelectedPulse" := "hmi".model[5];
   #_w6 := "hmi".model[6] AND NOT "model06SelectedPulse";   // rising edge
   "model06SelectedPulse" := "hmi".model[6];
   #_w7 := "hmi".model[7] AND NOT "model07SelectedPulse";   // rising edge
   "model07SelectedPulse" := "hmi".model[7];
   #_w8 := "hmi".model[8] AND NOT "model08SelectedPulse";   // rising edge
   "model08SelectedPulse" := "hmi".model[8];
   #_w9 := "hmi".model[9] AND NOT "model09SelectedPulse";   // rising edge
   "model09SelectedPulse" := "hmi".model[9];
   #_w10 := "hmi".model[10] AND NOT "model10SelectedPulse";   // rising edge
   "model10SelectedPulse" := "hmi".model[10];
   #_w11 := "hmi".model[11] AND NOT "model11SelectedPulse";   // rising edge
   "model11SelectedPulse" := "hmi".model[11];
   #_w12 := "hmi".model[12] AND NOT "model12SelectedPulse";   // rising edge
   "model12SelectedPulse" := "hmi".model[12];
   #_w13 := "hmi".model[13] AND NOT "model13SelectedPulse";   // rising edge
   "model13SelectedPulse" := "hmi".model[13];
   #_w14 := "hmi".model[14] AND NOT "model14SelectedPulse";   // rising edge
   "model14SelectedPulse" := "hmi".model[14];
   #_w15 := "hmi".model[15] AND NOT "model15SelectedPulse";   // rising edge
   "model15SelectedPulse" := "hmi".model[15];
   #_w16 := "hmi".model[16] AND NOT "model16SelectedPulse";   // rising edge
   "model16SelectedPulse" := "hmi".model[16];
   #_w17 := "hmi".model[17] AND NOT "model17SelectedPulse";   // rising edge
   "model17SelectedPulse" := "hmi".model[17];
   #_w18 := "hmi".model[18] AND NOT "model18SelectedPulse";   // rising edge
   "model18SelectedPulse" := "hmi".model[18];
   #_w19 := "hmi".model[19] AND NOT "model19SelectedPulse";   // rising edge
   "model19SelectedPulse" := "hmi".model[19];
   #_w20 := "hmi".model[20] AND NOT "model20SelectedPulse";   // rising edge
   "model20SelectedPulse" := "hmi".model[20];
   #_w21 := "hmi".model[21] AND NOT "model21SelectedPulse";   // rising edge
   "model21SelectedPulse" := "hmi".model[21];
   #_w22 := "hmi".model[22] AND NOT "model22SelectedPulse";   // rising edge
   "model22SelectedPulse" := "hmi".model[22];
   #_w23 := "hmi".model[23] AND NOT "model23SelectedPulse";   // rising edge
   "model23SelectedPulse" := "hmi".model[23];
   #_w24 := "hmi".model[24] AND NOT "model24SelectedPulse";   // rising edge
   "model24SelectedPulse" := "hmi".model[24];
   #_w25 := "hmi".model[25] AND NOT "model25SelectedPulse";   // rising edge
   "model25SelectedPulse" := "hmi".model[25];
   #_w26 := "hmi".model[26] AND NOT "model26SelectedPulse";   // rising edge
   "model26SelectedPulse" := "hmi".model[26];
   #_w27 := "hmi".model[27] AND NOT "model27SelectedPulse";   // rising edge
   "model27SelectedPulse" := "hmi".model[27];
   #_w28 := "hmi".model[28] AND NOT "model28SelectedPulse";   // rising edge
   "model28SelectedPulse" := "hmi".model[28];
   #_w29 := "hmi".model[29] AND NOT "model29SelectedPulse";   // rising edge
   "model29SelectedPulse" := "hmi".model[29];
   #_w30 := "hmi".model[30] AND NOT "model30SelectedPulse";   // rising edge
   "model30SelectedPulse" := "hmi".model[30];
   #_w31 := "hmi".model[31] AND NOT "model31SelectedPulse";   // rising edge
   "model31SelectedPulse" := "hmi".model[31];
   #_w32 := "hmi".model[32] AND NOT "model32SelectedPulse";   // rising edge
   "model32SelectedPulse" := "hmi".model[32];
   "hmi".modelChange := #_w1 OR #_w2 OR #_w3 OR #_w4 OR #_w5 OR #_w6 OR #_w7 OR #_w8 OR #_w9 OR #_w10 OR #_w11 OR #_w12 OR #_w13 OR #_w14 OR #_w15 OR #_w16 OR #_w17 OR #_w18 OR #_w19 OR #_w20 OR #_w21 OR #_w22 OR #_w23 OR #_w24 OR #_w25 OR #_w26 OR #_w27 OR #_w28 OR #_w29 OR #_w30 OR #_w31 OR #_w32;
END_REGION
END_FUNCTION

FUNCTION "dcMotorControl" : Void   // FC20, LAD
{ S7_Optimized_Access := 'TRUE' }
VERSION : 0.1
// stored: AutoNumber true, IsIECCheckEnabled false, SetENOAutomatically false, UDAEnableTagReadback false
   VAR_TEMP   // added for the SCL form of the ladder/FBD networks
      _w1 : Bool;
      _w2 : Bool;
   END_VAR
BEGIN

REGION Network 1: SELECT MOTOR PARAMETERS
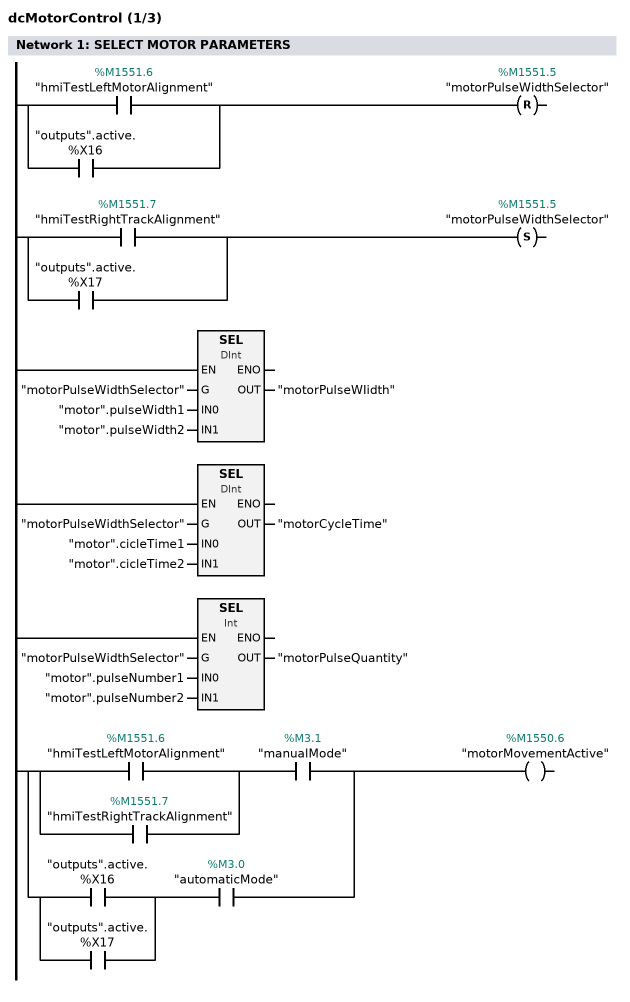
   RUNG wire#powerrail
      Contact( "hmiTestLeftMotorAlignment" )
      wire#w1
      R_Coil( "motorPulseWidthSelector" )
   END_RUNG
   RUNG wire#powerrail
      Contact( "outputs".active.%X16 )
   END_RUNG wire#w1
   RUNG wire#powerrail
      Contact( "hmiTestRightTrackAlignment" )
      wire#w2
      S_Coil( "motorPulseWidthSelector" )
   END_RUNG
   RUNG wire#powerrail
      Contact( "outputs".active.%X17 )
   END_RUNG wire#w2
   RUNG wire#powerrail
      { S7_Templates := "value_type := DInt" } SEL(g := "motorPulseWidthSelector", in0 := "motor".pulseWidth1, in1 := "motor".pulseWidth2, out => "motorPulseWIidth")
   END_RUNG
   RUNG wire#powerrail
      { S7_Templates := "value_type := DInt" } SEL(g := "motorPulseWidthSelector", in0 := "motor".cicleTime1, in1 := "motor".cicleTime2, out => "motorCycleTime")
   END_RUNG
   RUNG wire#powerrail
      { S7_Templates := "value_type := Int" } SEL(g := "motorPulseWidthSelector", in0 := "motor".pulseNumber1, in1 := "motor".pulseNumber2, out => "motorPulseQuantity")
   END_RUNG
   RUNG wire#powerrail
      Contact( "hmiTestLeftMotorAlignment" )
      wire#w3
      Contact( "manualMode" )
      wire#w4
      Coil( "motorMovementActive" )
   END_RUNG
   RUNG wire#powerrail
      Contact( "hmiTestRightTrackAlignment" )
   END_RUNG wire#w3
   RUNG wire#powerrail
      Contact( "outputs".active.%X16 )
      wire#w5
      Contact( "automaticMode" )
   END_RUNG wire#w4
   RUNG wire#powerrail
      Contact( "outputs".active.%X17 )
   END_RUNG wire#w5
   // the same network as SCL:
   IF "hmiTestLeftMotorAlignment" OR "outputs".active.%X16 THEN "motorPulseWidthSelector" := FALSE; END_IF;
   IF "hmiTestRightTrackAlignment" OR "outputs".active.%X17 THEN "motorPulseWidthSelector" := TRUE; END_IF;
   "motorPulseWIidth" := SEL(G := "motorPulseWidthSelector", IN0 := "motor".pulseWidth1, IN1 := "motor".pulseWidth2);
   "motorCycleTime" := SEL(G := "motorPulseWidthSelector", IN0 := "motor".cicleTime1, IN1 := "motor".cicleTime2);
   "motorPulseQuantity" := SEL(G := "motorPulseWidthSelector", IN0 := "motor".pulseNumber1, IN1 := "motor".pulseNumber2);
   "motorMovementActive" := (("hmiTestLeftMotorAlignment" OR "hmiTestRightTrackAlignment") AND "manualMode") OR (("outputs".active.%X16 OR "outputs".active.%X17) AND "automaticMode");
END_REGION

REGION Network 2: PWM CONTROL
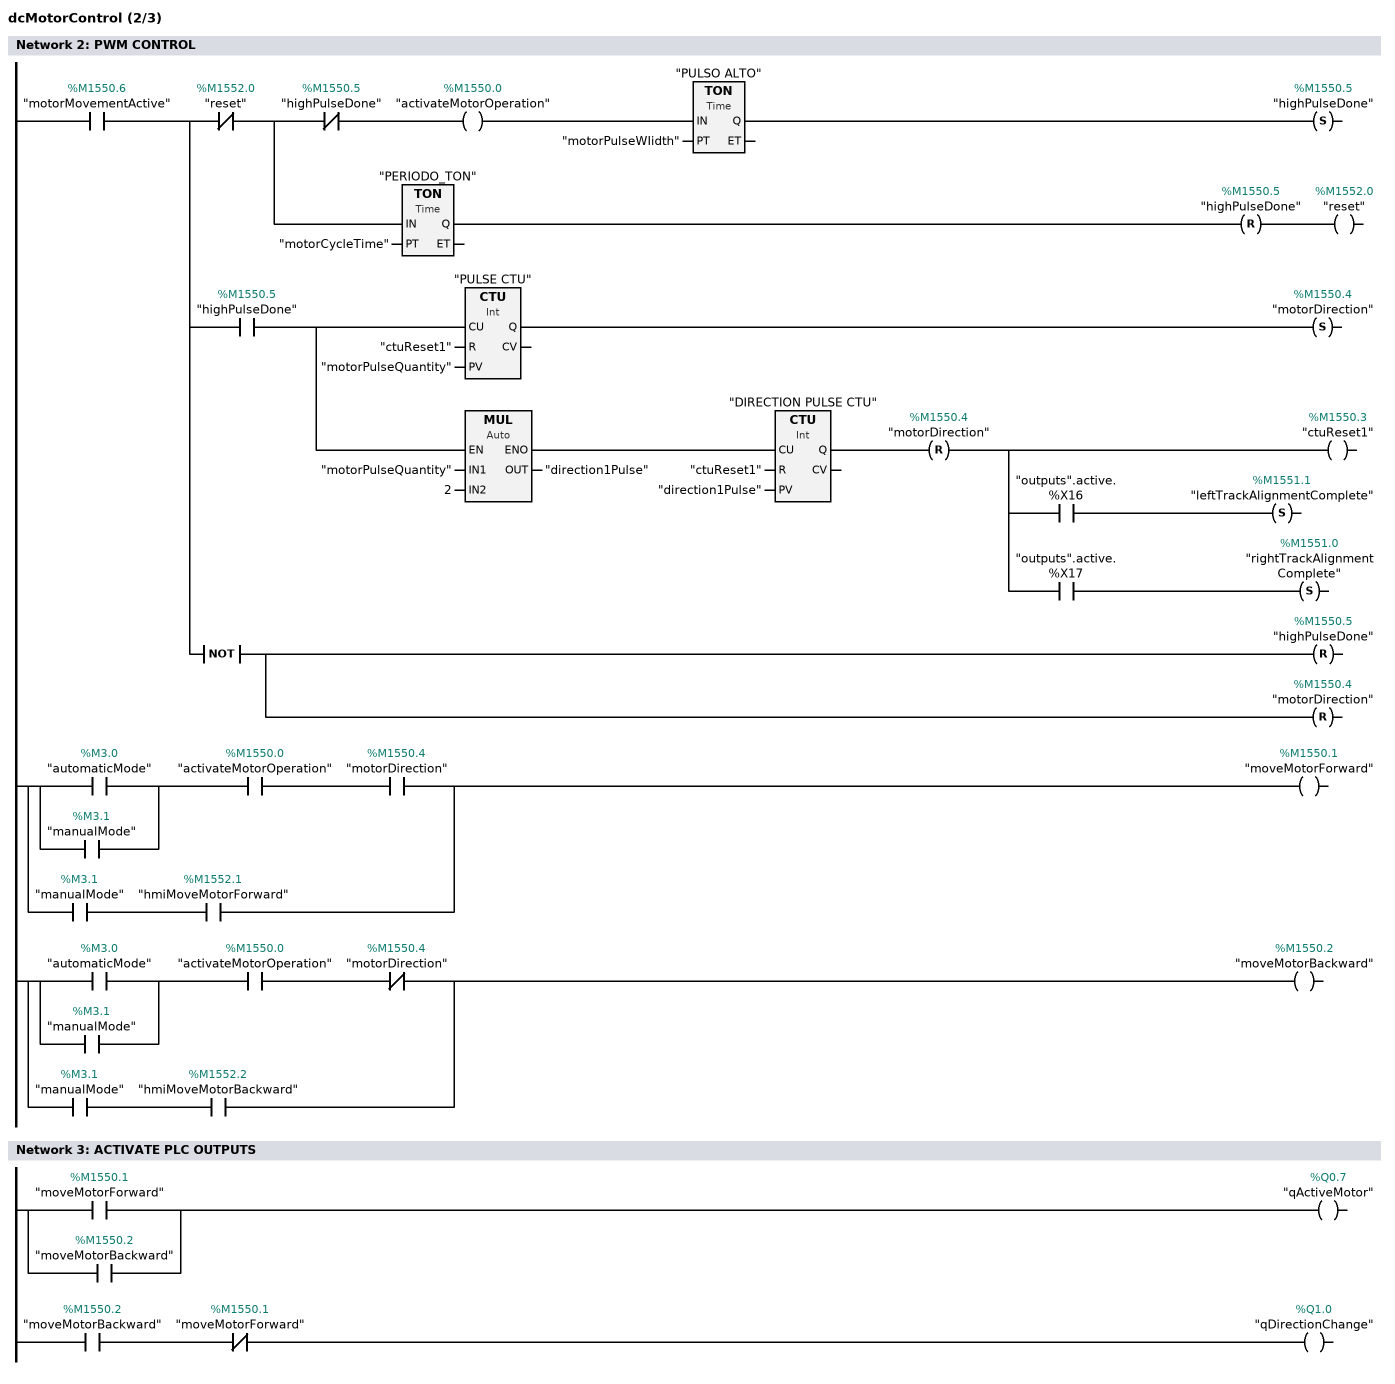
   RUNG wire#powerrail
      Contact( "motorMovementActive" )
      wire#w1
      I_Contact( "reset" )
      wire#w2
      I_Contact( "highPulseDone" )
      Coil( "activateMotorOperation" )
      { S7_Templates := "time_type := Time" } "PULSO ALTO".TON(pt := "motorPulseWIidth", et =>)
      S_Coil( "highPulseDone" )
   END_RUNG
   RUNG wire#w2
      { S7_Templates := "time_type := Time" } "PERIODO_TON".TON(pt := "motorCycleTime", et =>)
      R_Coil( "highPulseDone" )
      Coil( "reset" )
   END_RUNG
   RUNG wire#w1
      Contact( "highPulseDone" )
      wire#w3
      { S7_Templates := "value_type := Int" } "PULSE CTU".CTU(r := "ctuReset1", pv := "motorPulseQuantity", cv =>)
      S_Coil( "motorDirection" )
   END_RUNG
   RUNG wire#w3
      Mul(in1 := "motorPulseQuantity", in2 := 2, out => "direction1Pulse")
      { S7_Templates := "value_type := Int" } "DIRECTION PULSE CTU".CTU(r := "ctuReset1", pv := "direction1Pulse", cv =>)
      R_Coil( "motorDirection" )
      wire#w4
      Coil( "ctuReset1" )
   END_RUNG
   RUNG wire#w4
      Contact( "outputs".active.%X16 )
      S_Coil( "leftTrackAlignmentComplete" )
   END_RUNG
   RUNG wire#w4
      Contact( "outputs".active.%X17 )
      S_Coil( "rightTrackAlignmentComplete" )
   END_RUNG
   RUNG wire#w1
      Not()
      wire#w5
      R_Coil( "highPulseDone" )
   END_RUNG
   RUNG wire#w5
      R_Coil( "motorDirection" )
   END_RUNG
   RUNG wire#powerrail
      Contact( "automaticMode" )
      wire#w6
      Contact( "activateMotorOperation" )
      Contact( "motorDirection" )
      wire#w7
      Coil( "moveMotorForward" )
   END_RUNG
   RUNG wire#powerrail
      Contact( "manualMode" )
   END_RUNG wire#w6
   RUNG wire#powerrail
      Contact( "manualMode" )
      Contact( "hmiMoveMotorForward" )
   END_RUNG wire#w7
   RUNG wire#powerrail
      Contact( "automaticMode" )
      wire#w8
      Contact( "activateMotorOperation" )
      I_Contact( "motorDirection" )
      wire#w9
      Coil( "moveMotorBackward" )
   END_RUNG
   RUNG wire#powerrail
      Contact( "manualMode" )
   END_RUNG wire#w8
   RUNG wire#powerrail
      Contact( "manualMode" )
      Contact( "hmiMoveMotorBackward" )
   END_RUNG wire#w9
   // the same network as SCL:
   #_w1 := "motorMovementActive" AND NOT "reset";
   "activateMotorOperation" := #_w1 AND NOT "highPulseDone";
   "PULSO ALTO".TON(IN := "activateMotorOperation", PT := "motorPulseWIidth");
   IF "PULSO ALTO".Q THEN "highPulseDone" := TRUE; END_IF;
   "PERIODO_TON".TON(IN := #_w1, PT := "motorCycleTime");
   IF "PERIODO_TON".Q THEN "highPulseDone" := FALSE; END_IF;
   "reset" := "PERIODO_TON".Q;
   #_w2 := "motorMovementActive" AND "highPulseDone";
   "PULSE CTU".CTU(CU := #_w2, R := "ctuReset1", PV := "motorPulseQuantity");
   IF "PULSE CTU".Q THEN "motorDirection" := TRUE; END_IF;
   IF #_w2 THEN "direction1Pulse" := "motorPulseQuantity" * 2; END_IF;
   "DIRECTION PULSE CTU".CTU(CU := #_w2, R := "ctuReset1", PV := "direction1Pulse");
   IF "DIRECTION PULSE CTU".Q THEN "motorDirection" := FALSE; END_IF;
   "ctuReset1" := "DIRECTION PULSE CTU".Q;
   IF "DIRECTION PULSE CTU".Q AND "outputs".active.%X16 THEN "leftTrackAlignmentComplete" := TRUE; END_IF;
   IF "DIRECTION PULSE CTU".Q AND "outputs".active.%X17 THEN "rightTrackAlignmentComplete" := TRUE; END_IF;
   IF NOT "motorMovementActive" THEN
       "highPulseDone" := FALSE;
       "motorDirection" := FALSE;
   END_IF;
   "moveMotorForward" := (("automaticMode" OR "manualMode") AND "activateMotorOperation" AND "motorDirection") OR ("manualMode" AND "hmiMoveMotorForward");
   "moveMotorBackward" := (("automaticMode" OR "manualMode") AND "activateMotorOperation" AND NOT "motorDirection") OR ("manualMode" AND "hmiMoveMotorBackward");
END_REGION

REGION Network 3: ACTIVATE PLC OUTPUTS
   RUNG wire#powerrail
      Contact( "moveMotorForward" )
      wire#w1
      Coil( "qActiveMotor" )
   END_RUNG
   RUNG wire#powerrail
      Contact( "moveMotorBackward" )
   END_RUNG wire#w1
   RUNG wire#powerrail
      Contact( "moveMotorBackward" )
      I_Contact( "moveMotorForward" )
      Coil( "qDirectionChange" )
   END_RUNG
   // the same network as SCL:
   "qActiveMotor" := "moveMotorForward" OR "moveMotorBackward";
   "qDirectionChange" := "moveMotorBackward" AND NOT "moveMotorForward";
END_REGION

REGION Network 4: RESET SEQUENCER STATUS
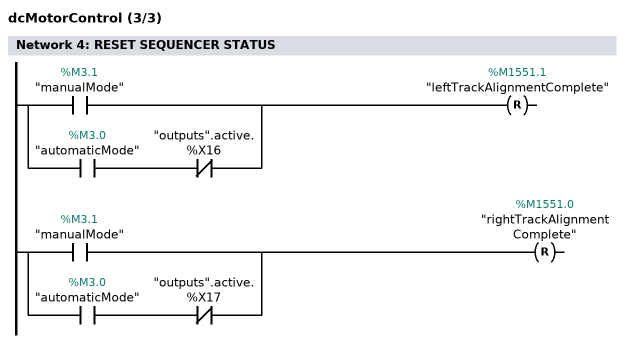
   RUNG wire#powerrail
      Contact( "manualMode" )
      wire#w1
      R_Coil( "leftTrackAlignmentComplete" )
   END_RUNG
   RUNG wire#powerrail
      Contact( "automaticMode" )
      I_Contact( "outputs".active.%X16 )
   END_RUNG wire#w1
   RUNG wire#powerrail
      Contact( "manualMode" )
      wire#w2
      R_Coil( "rightTrackAlignmentComplete" )
   END_RUNG
   RUNG wire#powerrail
      Contact( "automaticMode" )
      I_Contact( "outputs".active.%X17 )
   END_RUNG wire#w2
   // the same network as SCL:
   IF "manualMode" OR ("automaticMode" AND NOT "outputs".active.%X16) THEN
       "leftTrackAlignmentComplete" := FALSE;
   END_IF;
   IF "manualMode" OR ("automaticMode" AND NOT "outputs".active.%X17) THEN
       "rightTrackAlignmentComplete" := FALSE;
   END_IF;
END_REGION
END_FUNCTION

FUNCTION "analogSignals" : Void   // FC16, LAD
{ S7_Optimized_Access := 'TRUE' }
VERSION : 0.1
// stored: AutoNumber true, IsIECCheckEnabled false, SetENOAutomatically false, UDAEnableTagReadback false
   VAR_TEMP
      minimumScaleRangeArray : Array[0..9] of Real;
      maximumScaleRangeArray : Array[0..9] of Real;
      i : Int;
   END_VAR
BEGIN

REGION Network 1 (SCL): Initialize Temp Values
   FOR #i := 0 TO 9 DO
       #minimumScaleRangeArray[#i] := 0;
       #maximumScaleRangeArray[#i] := 0;
   END_FOR;
END_REGION

REGION Network 2: Load Cell Adquisition
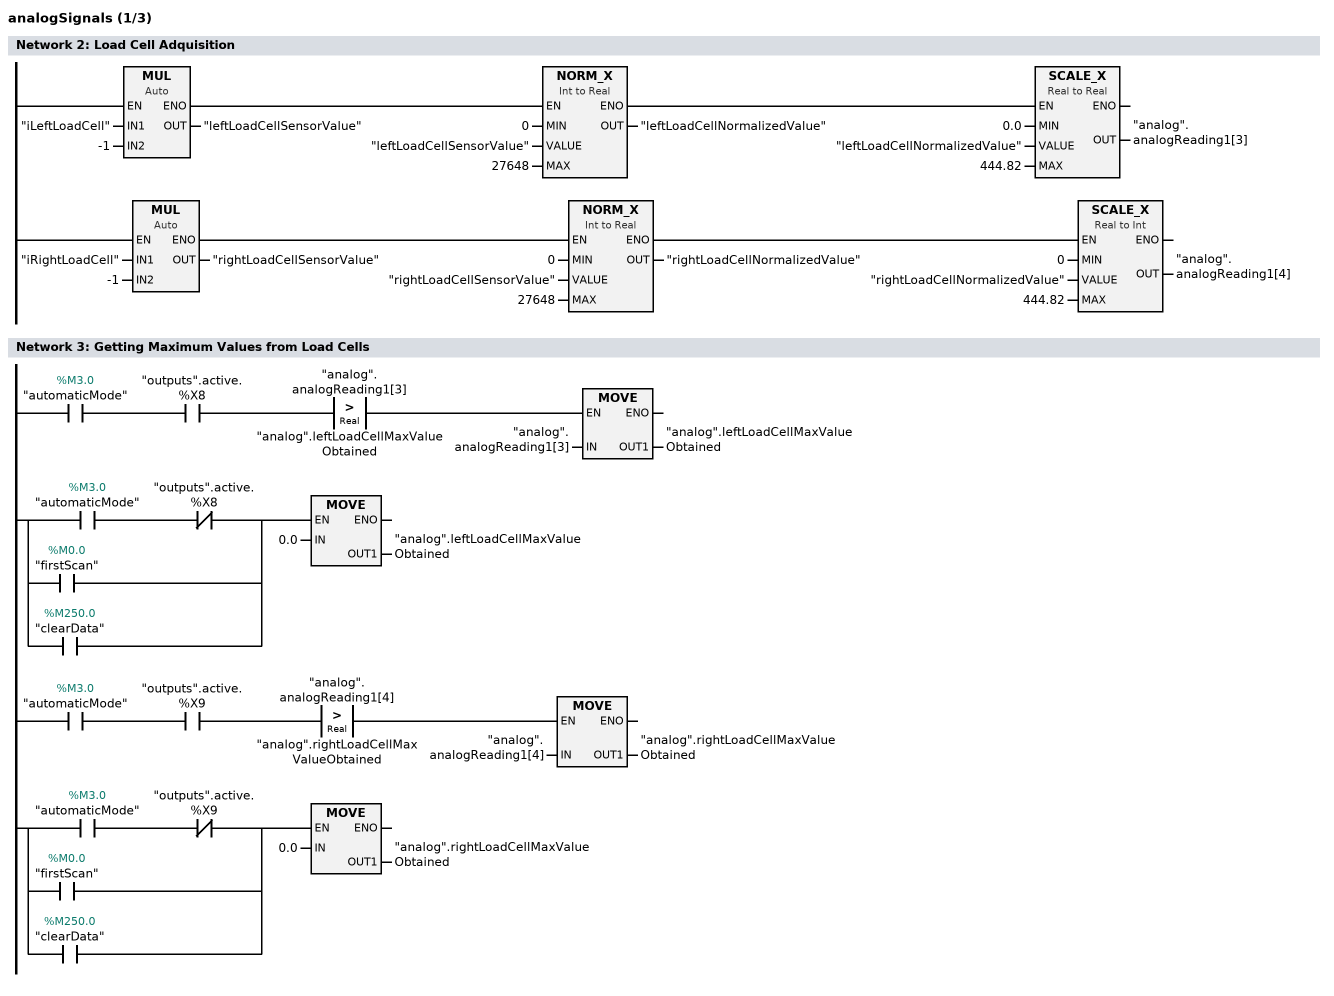
   RUNG wire#powerrail
      Mul(in1 := "iLeftLoadCell", in2 := -1, out => "leftLoadCellSensorValue")
      { S7_Templates := "[SrcType := Int, DestType := Real]" } Normalize(min := 0, value := "leftLoadCellSensorValue", max := 27648, out => "leftLoadCellNormalizedValue")
      { S7_Templates := "[SrcType := Real, DestType := Real]" } Scale(min := 0.0, value := "leftLoadCellNormalizedValue", max := 444.82, out => "analog".analogReading1[3])
   END_RUNG
   RUNG wire#powerrail
      Mul(in1 := "iRightLoadCell", in2 := -1, out => "rightLoadCellSensorValue")
      { S7_Templates := "[SrcType := Int, DestType := Real]" } Normalize(min := 0, value := "rightLoadCellSensorValue", max := 27648, out => "rightLoadCellNormalizedValue")
      { S7_Templates := "[SrcType := Real, DestType := Int]" } Scale(min := 0, value := "rightLoadCellNormalizedValue", max := 444.82, out => "analog".analogReading1[4])
   END_RUNG
   // the same network as SCL:
   "leftLoadCellSensorValue" := "iLeftLoadCell" * (-1);
   "leftLoadCellNormalizedValue" := NORM_X(MIN := 0, VALUE := "leftLoadCellSensorValue", MAX := 27648);
   "analog".analogReading1[3] := SCALE_X(MIN := 0.0, VALUE := "leftLoadCellNormalizedValue", MAX := 444.82);
   "rightLoadCellSensorValue" := "iRightLoadCell" * (-1);
   "rightLoadCellNormalizedValue" := NORM_X(MIN := 0, VALUE := "rightLoadCellSensorValue", MAX := 27648);
   "analog".analogReading1[4] := SCALE_X(MIN := 0, VALUE := "rightLoadCellNormalizedValue", MAX := 444.82);
END_REGION

REGION Network 3: Getting Maximum Values from Load Cells
   RUNG wire#powerrail
      Contact( "automaticMode" )
      Contact( "outputs".active.%X8 )
      { S7_Templates := "SrcType := Real" } GT_Contact(in1 := "analog".analogReading1[3], in2 := "analog".leftLoadCellMaxValueObtained)
      Move(in := "analog".analogReading1[3], out1 => "analog".leftLoadCellMaxValueObtained)
   END_RUNG
   RUNG wire#powerrail
      Contact( "automaticMode" )
      I_Contact( "outputs".active.%X8 )
      wire#w1
      Move(in := 0.0, out1 => "analog".leftLoadCellMaxValueObtained)
   END_RUNG
   RUNG wire#powerrail
      Contact( "firstScan" )
   END_RUNG wire#w1
   RUNG wire#powerrail
      Contact( "clearData" )
   END_RUNG wire#w1
   RUNG wire#powerrail
      Contact( "automaticMode" )
      Contact( "outputs".active.%X9 )
      { S7_Templates := "SrcType := Real" } GT_Contact(in1 := "analog".analogReading1[4], in2 := "analog".rightLoadCellMaxValueObtained)
      Move(in := "analog".analogReading1[4], out1 => "analog".rightLoadCellMaxValueObtained)
   END_RUNG
   RUNG wire#powerrail
      Contact( "automaticMode" )
      I_Contact( "outputs".active.%X9 )
      wire#w2
      Move(in := 0.0, out1 => "analog".rightLoadCellMaxValueObtained)
   END_RUNG
   RUNG wire#powerrail
      Contact( "firstScan" )
   END_RUNG wire#w2
   RUNG wire#powerrail
      Contact( "clearData" )
   END_RUNG wire#w2
   // the same network as SCL:
   IF "automaticMode" AND "outputs".active.%X8 AND ("analog".analogReading1[3] > "analog".leftLoadCellMaxValueObtained) THEN
       "analog".leftLoadCellMaxValueObtained := "analog".analogReading1[3];
   END_IF;
   IF ("automaticMode" AND NOT "outputs".active.%X8) OR "firstScan" OR "clearData" THEN
       "analog".leftLoadCellMaxValueObtained := 0.0;
   END_IF;
   IF "automaticMode" AND "outputs".active.%X9 AND ("analog".analogReading1[4] > "analog".rightLoadCellMaxValueObtained) THEN
       "analog".rightLoadCellMaxValueObtained := "analog".analogReading1[4];
   END_IF;
   IF ("automaticMode" AND NOT "outputs".active.%X9) OR "firstScan" OR "clearData" THEN
       "analog".rightLoadCellMaxValueObtained := 0.0;
   END_IF;
END_REGION

REGION Network 4: Effort OK/NOK Evaluation
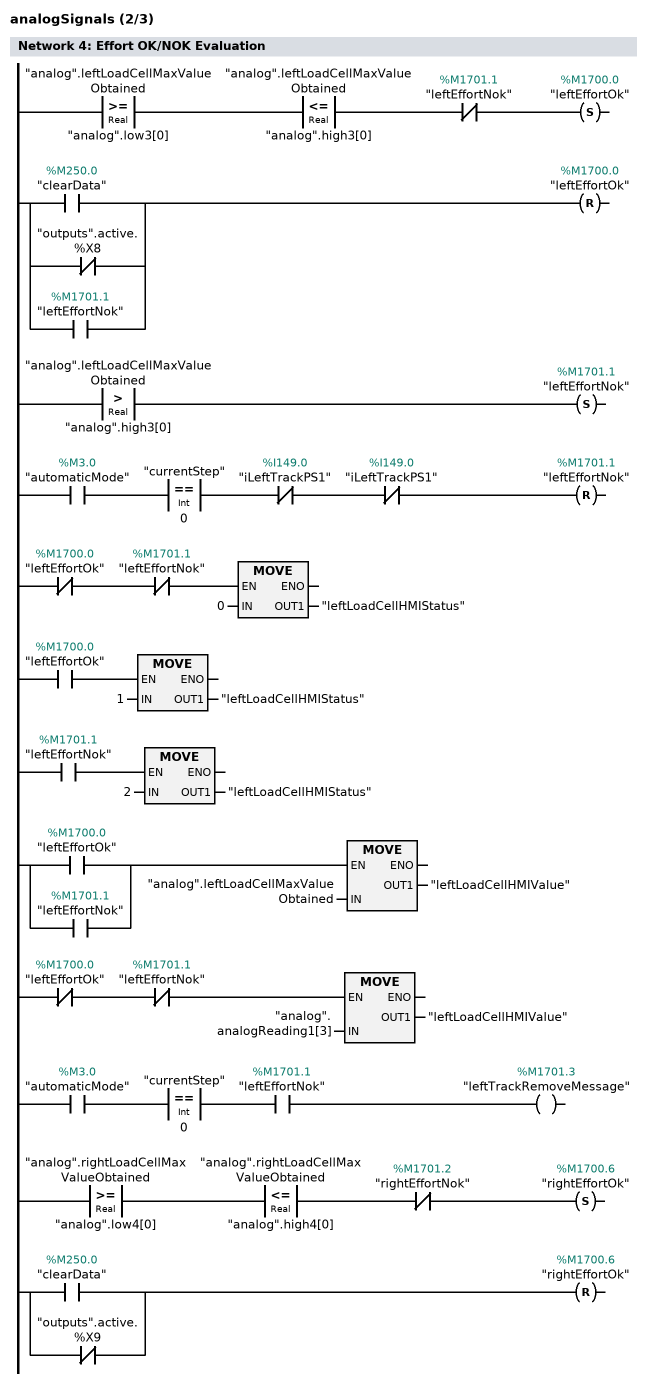
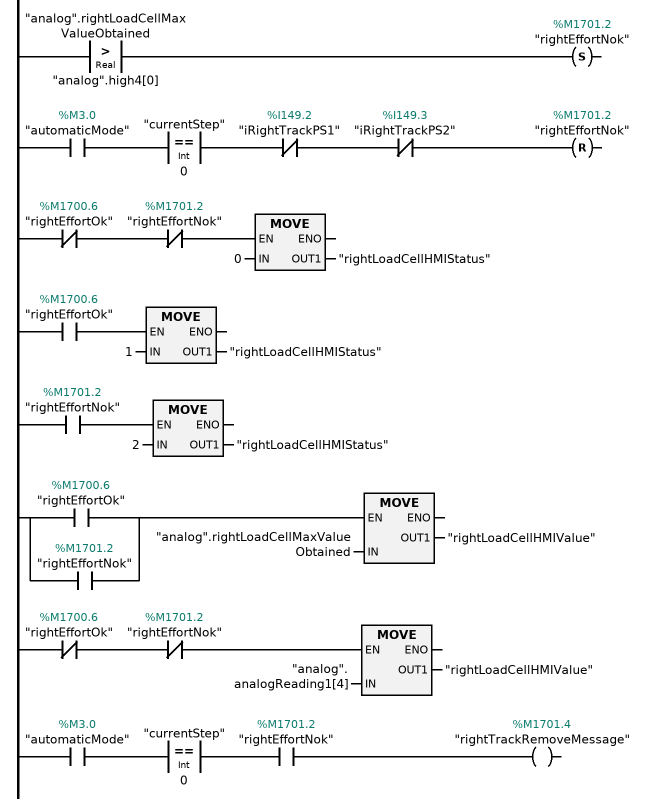
   RUNG wire#powerrail
      { S7_Templates := "SrcType := Real" } GE_Contact(in1 := "analog".leftLoadCellMaxValueObtained, in2 := "analog".low3[0])
      { S7_Templates := "SrcType := Real" } LE_Contact(in1 := "analog".leftLoadCellMaxValueObtained, in2 := "analog".high3[0])
      I_Contact( "leftEffortNok" )
      S_Coil( "leftEffortOk" )
   END_RUNG
   RUNG wire#powerrail
      Contact( "clearData" )
      wire#w1
      R_Coil( "leftEffortOk" )
   END_RUNG
   RUNG wire#powerrail
      I_Contact( "outputs".active.%X8 )
   END_RUNG wire#w1
   RUNG wire#powerrail
      Contact( "leftEffortNok" )
   END_RUNG wire#w1
   RUNG wire#powerrail
      { S7_Templates := "SrcType := Real" } GT_Contact(in1 := "analog".leftLoadCellMaxValueObtained, in2 := "analog".high3[0])
      S_Coil( "leftEffortNok" )
   END_RUNG
   RUNG wire#powerrail
      Contact( "automaticMode" )
      { S7_Templates := "SrcType := Int" } EQ_Contact(in1 := "currentStep", in2 := 0)
      I_Contact( "iLeftTrackPS1" )
      I_Contact( "iLeftTrackPS1" )
      R_Coil( "leftEffortNok" )
   END_RUNG
   RUNG wire#powerrail
      I_Contact( "leftEffortOk" )
      I_Contact( "leftEffortNok" )
      Move(in := 0, out1 => "leftLoadCellHMIStatus")
   END_RUNG
   RUNG wire#powerrail
      Contact( "leftEffortOk" )
      Move(in := 1, out1 => "leftLoadCellHMIStatus")
   END_RUNG
   RUNG wire#powerrail
      Contact( "leftEffortNok" )
      Move(in := 2, out1 => "leftLoadCellHMIStatus")
   END_RUNG
   RUNG wire#powerrail
      Contact( "leftEffortOk" )
      wire#w2
      Move(in := "analog".leftLoadCellMaxValueObtained, out1 => "leftLoadCellHMIValue")
   END_RUNG
   RUNG wire#powerrail
      Contact( "leftEffortNok" )
   END_RUNG wire#w2
   RUNG wire#powerrail
      I_Contact( "leftEffortOk" )
      I_Contact( "leftEffortNok" )
      Move(in := "analog".analogReading1[3], out1 => "leftLoadCellHMIValue")
   END_RUNG
   RUNG wire#powerrail
      Contact( "automaticMode" )
      { S7_Templates := "SrcType := Int" } EQ_Contact(in1 := "currentStep", in2 := 0)
      Contact( "leftEffortNok" )
      Coil( "leftTrackRemoveMessage" )
   END_RUNG
   RUNG wire#powerrail
      { S7_Templates := "SrcType := Real" } GE_Contact(in1 := "analog".rightLoadCellMaxValueObtained, in2 := "analog".low4[0])
      { S7_Templates := "SrcType := Real" } LE_Contact(in1 := "analog".rightLoadCellMaxValueObtained, in2 := "analog".high4[0])
      I_Contact( "rightEffortNok" )
      S_Coil( "rightEffortOk" )
   END_RUNG
   RUNG wire#powerrail
      Contact( "clearData" )
      wire#w3
      R_Coil( "rightEffortOk" )
   END_RUNG
   RUNG wire#powerrail
      I_Contact( "outputs".active.%X9 )
   END_RUNG wire#w3
   RUNG wire#powerrail
      { S7_Templates := "SrcType := Real" } GT_Contact(in1 := "analog".rightLoadCellMaxValueObtained, in2 := "analog".high4[0])
      S_Coil( "rightEffortNok" )
   END_RUNG
   RUNG wire#powerrail
      Contact( "automaticMode" )
      { S7_Templates := "SrcType := Int" } EQ_Contact(in1 := "currentStep", in2 := 0)
      I_Contact( "iRightTrackPS1" )
      I_Contact( "iRightTrackPS2" )
      R_Coil( "rightEffortNok" )
   END_RUNG
   RUNG wire#powerrail
      I_Contact( "rightEffortOk" )
      I_Contact( "rightEffortNok" )
      Move(in := 0, out1 => "rightLoadCellHMIStatus")
   END_RUNG
   RUNG wire#powerrail
      Contact( "rightEffortOk" )
      Move(in := 1, out1 => "rightLoadCellHMIStatus")
   END_RUNG
   RUNG wire#powerrail
      Contact( "rightEffortNok" )
      Move(in := 2, out1 => "rightLoadCellHMIStatus")
   END_RUNG
   RUNG wire#powerrail
      Contact( "rightEffortOk" )
      wire#w4
      Move(in := "analog".rightLoadCellMaxValueObtained, out1 => "rightLoadCellHMIValue")
   END_RUNG
   RUNG wire#powerrail
      Contact( "rightEffortNok" )
   END_RUNG wire#w4
   RUNG wire#powerrail
      I_Contact( "rightEffortOk" )
      I_Contact( "rightEffortNok" )
      Move(in := "analog".analogReading1[4], out1 => "rightLoadCellHMIValue")
   END_RUNG
   RUNG wire#powerrail
      Contact( "automaticMode" )
      { S7_Templates := "SrcType := Int" } EQ_Contact(in1 := "currentStep", in2 := 0)
      Contact( "rightEffortNok" )
      Coil( "rightTrackRemoveMessage" )
   END_RUNG
   // the same network as SCL:
   IF ("analog".leftLoadCellMaxValueObtained >= "analog".low3[0]) AND ("analog".leftLoadCellMaxValueObtained <= "analog".high3[0]) AND NOT "leftEffortNok" THEN
       "leftEffortOk" := TRUE;
   END_IF;
   IF "clearData" OR NOT "outputs".active.%X8 OR "leftEffortNok" THEN "leftEffortOk" := FALSE; END_IF;
   IF "analog".leftLoadCellMaxValueObtained > "analog".high3[0] THEN "leftEffortNok" := TRUE; END_IF;
   IF "automaticMode" AND ("currentStep" = 0) AND NOT "iLeftTrackPS1" AND NOT "iLeftTrackPS1" THEN
       "leftEffortNok" := FALSE;
   END_IF;
   IF NOT "leftEffortOk" AND NOT "leftEffortNok" THEN "leftLoadCellHMIStatus" := 0; END_IF;
   IF "leftEffortOk" THEN "leftLoadCellHMIStatus" := 1; END_IF;
   IF "leftEffortNok" THEN "leftLoadCellHMIStatus" := 2; END_IF;
   IF "leftEffortOk" OR "leftEffortNok" THEN
       "leftLoadCellHMIValue" := "analog".leftLoadCellMaxValueObtained;
   END_IF;
   IF NOT "leftEffortOk" AND NOT "leftEffortNok" THEN
       "leftLoadCellHMIValue" := "analog".analogReading1[3];
   END_IF;
   "leftTrackRemoveMessage" := "automaticMode" AND ("currentStep" = 0) AND "leftEffortNok";
   IF ("analog".rightLoadCellMaxValueObtained >= "analog".low4[0]) AND ("analog".rightLoadCellMaxValueObtained <= "analog".high4[0]) AND NOT "rightEffortNok" THEN
       "rightEffortOk" := TRUE;
   END_IF;
   IF "clearData" OR NOT "outputs".active.%X9 THEN "rightEffortOk" := FALSE; END_IF;
   IF "analog".rightLoadCellMaxValueObtained > "analog".high4[0] THEN "rightEffortNok" := TRUE; END_IF;
   IF "automaticMode" AND ("currentStep" = 0) AND NOT "iRightTrackPS1" AND NOT "iRightTrackPS2" THEN
       "rightEffortNok" := FALSE;
   END_IF;
   IF NOT "rightEffortOk" AND NOT "rightEffortNok" THEN "rightLoadCellHMIStatus" := 0; END_IF;
   IF "rightEffortOk" THEN "rightLoadCellHMIStatus" := 1; END_IF;
   IF "rightEffortNok" THEN "rightLoadCellHMIStatus" := 2; END_IF;
   IF "rightEffortOk" OR "rightEffortNok" THEN
       "rightLoadCellHMIValue" := "analog".rightLoadCellMaxValueObtained;
   END_IF;
   IF NOT "rightEffortOk" AND NOT "rightEffortNok" THEN
       "rightLoadCellHMIValue" := "analog".analogReading1[4];
   END_IF;
   "rightTrackRemoveMessage" := "automaticMode" AND ("currentStep" = 0) AND "rightEffortNok";
END_REGION

REGION Network 5: SENSOR DISTANCES
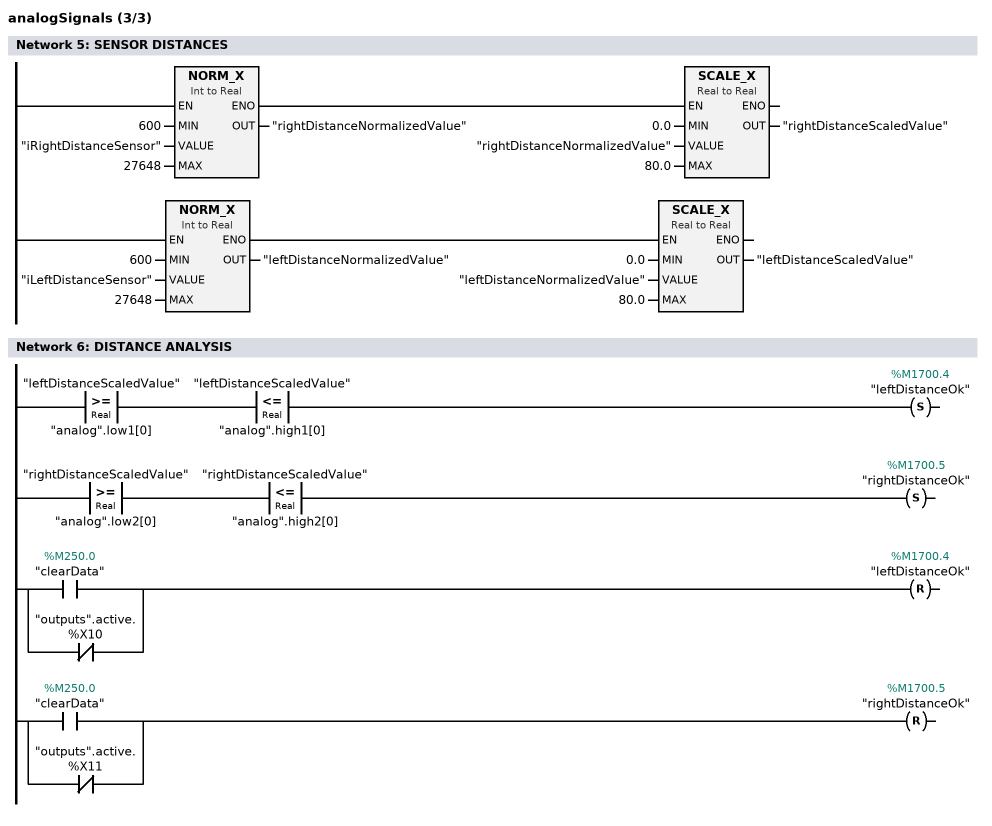
   RUNG wire#powerrail
      { S7_Templates := "[SrcType := Int, DestType := Real]" } Normalize(min := 600, value := "iRightDistanceSensor", max := 27648, out => "rightDistanceNormalizedValue")
      { S7_Templates := "[SrcType := Real, DestType := Real]" } Scale(min := 0.0, value := "rightDistanceNormalizedValue", max := 80.0, out => "rightDistanceScaledValue")
   END_RUNG
   RUNG wire#powerrail
      { S7_Templates := "[SrcType := Int, DestType := Real]" } Normalize(min := 600, value := "iLeftDistanceSensor", max := 27648, out => "leftDistanceNormalizedValue")
      { S7_Templates := "[SrcType := Real, DestType := Real]" } Scale(min := 0.0, value := "leftDistanceNormalizedValue", max := 80.0, out => "leftDistanceScaledValue")
   END_RUNG
   // the same network as SCL:
   "rightDistanceNormalizedValue" := NORM_X(MIN := 600, VALUE := "iRightDistanceSensor", MAX := 27648);
   "rightDistanceScaledValue" := SCALE_X(MIN := 0.0, VALUE := "rightDistanceNormalizedValue", MAX := 80.0);
   "leftDistanceNormalizedValue" := NORM_X(MIN := 600, VALUE := "iLeftDistanceSensor", MAX := 27648);
   "leftDistanceScaledValue" := SCALE_X(MIN := 0.0, VALUE := "leftDistanceNormalizedValue", MAX := 80.0);
END_REGION

REGION Network 6: DISTANCE ANALYSIS
   RUNG wire#powerrail
      { S7_Templates := "SrcType := Real" } GE_Contact(in1 := "leftDistanceScaledValue", in2 := "analog".low1[0])
      { S7_Templates := "SrcType := Real" } LE_Contact(in1 := "leftDistanceScaledValue", in2 := "analog".high1[0])
      S_Coil( "leftDistanceOk" )
   END_RUNG
   RUNG wire#powerrail
      { S7_Templates := "SrcType := Real" } GE_Contact(in1 := "rightDistanceScaledValue", in2 := "analog".low2[0])
      { S7_Templates := "SrcType := Real" } LE_Contact(in1 := "rightDistanceScaledValue", in2 := "analog".high2[0])
      S_Coil( "rightDistanceOk" )
   END_RUNG
   RUNG wire#powerrail
      Contact( "clearData" )
      wire#w1
      R_Coil( "leftDistanceOk" )
   END_RUNG
   RUNG wire#powerrail
      I_Contact( "outputs".active.%X10 )
   END_RUNG wire#w1
   RUNG wire#powerrail
      Contact( "clearData" )
      wire#w2
      R_Coil( "rightDistanceOk" )
   END_RUNG
   RUNG wire#powerrail
      I_Contact( "outputs".active.%X11 )
   END_RUNG wire#w2
   // the same network as SCL:
   IF ("leftDistanceScaledValue" >= "analog".low1[0]) AND ("leftDistanceScaledValue" <= "analog".high1[0]) THEN
       "leftDistanceOk" := TRUE;
   END_IF;
   IF ("rightDistanceScaledValue" >= "analog".low2[0]) AND ("rightDistanceScaledValue" <= "analog".high2[0]) THEN
       "rightDistanceOk" := TRUE;
   END_IF;
   IF "clearData" OR NOT "outputs".active.%X10 THEN "leftDistanceOk" := FALSE; END_IF;
   IF "clearData" OR NOT "outputs".active.%X11 THEN "rightDistanceOk" := FALSE; END_IF;
END_REGION
END_FUNCTION

FUNCTION "mode" : Void   // FC4, LAD
{ S7_Optimized_Access := 'TRUE' }
VERSION : 0.1
// stored: AutoNumber true, IsIECCheckEnabled false, SetENOAutomatically false, UDAEnableTagReadback false
   VAR_TEMP
      f7 : Bool;
      BF7 : Bool;
   END_VAR
BEGIN

REGION Network 1: MODE CHANGE
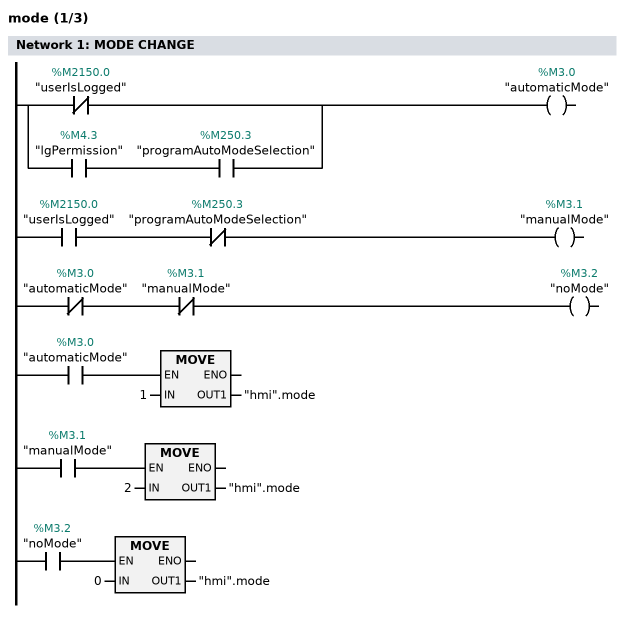
   RUNG wire#powerrail
      I_Contact( "userIsLogged" )
      wire#w1
      Coil( "automaticMode" )
   END_RUNG
   RUNG wire#powerrail
      Contact( "lgPermission" )
      Contact( "programAutoModeSelection" )
   END_RUNG wire#w1
   RUNG wire#powerrail
      Contact( "userIsLogged" )
      I_Contact( "programAutoModeSelection" )
      Coil( "manualMode" )
   END_RUNG
   RUNG wire#powerrail
      I_Contact( "automaticMode" )
      I_Contact( "manualMode" )
      Coil( "noMode" )
   END_RUNG
   RUNG wire#powerrail
      Contact( "automaticMode" )
      Move(in := 1, out1 => "hmi".mode)
   END_RUNG
   RUNG wire#powerrail
      Contact( "manualMode" )
      Move(in := 2, out1 => "hmi".mode)
   END_RUNG
   RUNG wire#powerrail
      Contact( "noMode" )
      Move(in := 0, out1 => "hmi".mode)
   END_RUNG
   // the same network as SCL:
   "automaticMode" := NOT "userIsLogged" OR ("lgPermission" AND "programAutoModeSelection");
   "manualMode" := "userIsLogged" AND NOT "programAutoModeSelection";
   "noMode" := NOT "automaticMode" AND NOT "manualMode";
   IF "automaticMode" THEN "hmi".mode := 1; END_IF;
   IF "manualMode" THEN "hmi".mode := 2; END_IF;
   IF "noMode" THEN "hmi".mode := 0; END_IF;
END_REGION

REGION Network 2: MODEL SELECTION
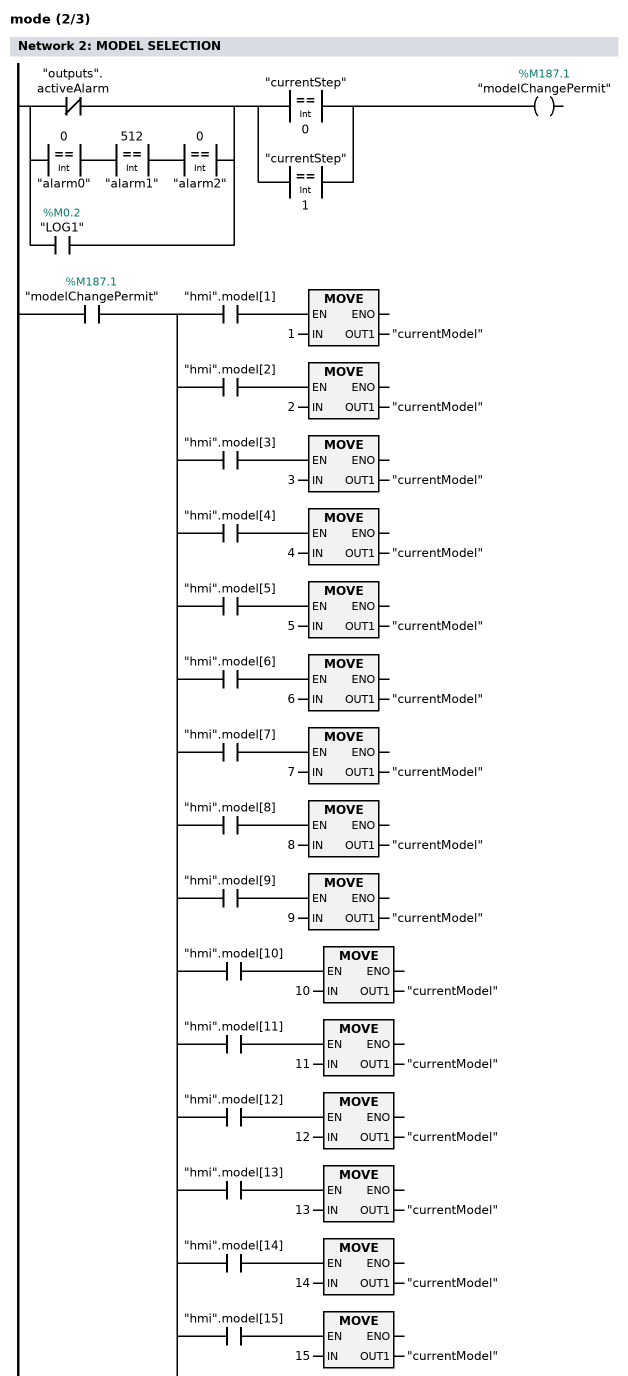
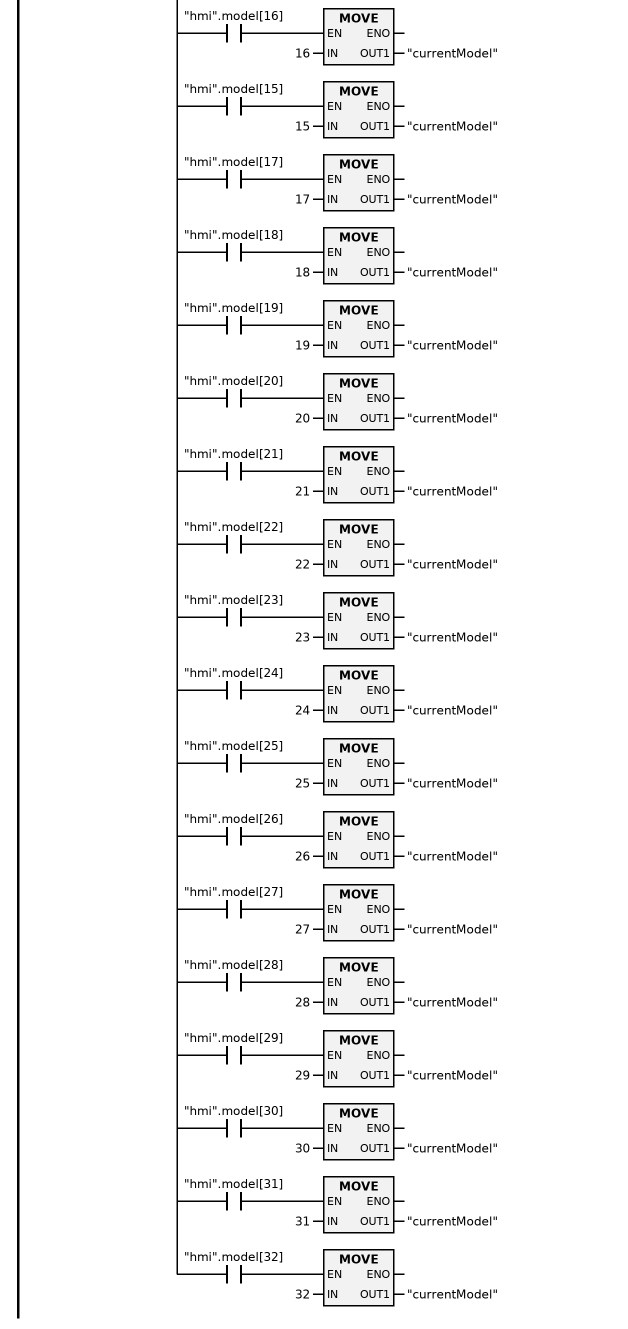
   RUNG wire#powerrail
      I_Contact( "outputs".activeAlarm )
      wire#w1
      { S7_Templates := "SrcType := Int" } EQ_Contact(in1 := "currentStep", in2 := 0)
      wire#w2
      Coil( "modelChangePermit" )
   END_RUNG
   RUNG wire#powerrail
      { S7_Templates := "SrcType := Int" } EQ_Contact(in1 := 0, in2 := "alarm0")
      { S7_Templates := "SrcType := Int" } EQ_Contact(in1 := 512, in2 := "alarm1")
      { S7_Templates := "SrcType := Int" } EQ_Contact(in1 := 0, in2 := "alarm2")
   END_RUNG wire#w1
   RUNG wire#powerrail
      Contact( "LOG1" )
   END_RUNG wire#w1
   RUNG wire#w1
      { S7_Templates := "SrcType := Int" } EQ_Contact(in1 := "currentStep", in2 := 1)
   END_RUNG wire#w2
   RUNG wire#powerrail
      Contact( "modelChangePermit" )
      wire#w3
      Contact( "hmi".model[1] )
      Move(in := 1, out1 => "currentModel")
   END_RUNG
   RUNG wire#w3
      Contact( "hmi".model[2] )
      Move(in := 2, out1 => "currentModel")
   END_RUNG
   RUNG wire#w3
      Contact( "hmi".model[3] )
      Move(in := 3, out1 => "currentModel")
   END_RUNG
   RUNG wire#w3
      Contact( "hmi".model[4] )
      Move(in := 4, out1 => "currentModel")
   END_RUNG
   RUNG wire#w3
      Contact( "hmi".model[5] )
      Move(in := 5, out1 => "currentModel")
   END_RUNG
   RUNG wire#w3
      Contact( "hmi".model[6] )
      Move(in := 6, out1 => "currentModel")
   END_RUNG
   RUNG wire#w3
      Contact( "hmi".model[7] )
      Move(in := 7, out1 => "currentModel")
   END_RUNG
   RUNG wire#w3
      Contact( "hmi".model[8] )
      Move(in := 8, out1 => "currentModel")
   END_RUNG
   RUNG wire#w3
      Contact( "hmi".model[9] )
      Move(in := 9, out1 => "currentModel")
   END_RUNG
   RUNG wire#w3
      Contact( "hmi".model[10] )
      Move(in := 10, out1 => "currentModel")
   END_RUNG
   RUNG wire#w3
      Contact( "hmi".model[11] )
      Move(in := 11, out1 => "currentModel")
   END_RUNG
   RUNG wire#w3
      Contact( "hmi".model[12] )
      Move(in := 12, out1 => "currentModel")
   END_RUNG
   RUNG wire#w3
      Contact( "hmi".model[13] )
      Move(in := 13, out1 => "currentModel")
   END_RUNG
   RUNG wire#w3
      Contact( "hmi".model[14] )
      Move(in := 14, out1 => "currentModel")
   END_RUNG
   RUNG wire#w3
      Contact( "hmi".model[15] )
      Move(in := 15, out1 => "currentModel")
   END_RUNG
   RUNG wire#w3
      Contact( "hmi".model[16] )
      Move(in := 16, out1 => "currentModel")
   END_RUNG
   RUNG wire#w3
      Contact( "hmi".model[15] )
      Move(in := 15, out1 => "currentModel")
   END_RUNG
   RUNG wire#w3
      Contact( "hmi".model[17] )
      Move(in := 17, out1 => "currentModel")
   END_RUNG
   RUNG wire#w3
      Contact( "hmi".model[18] )
      Move(in := 18, out1 => "currentModel")
   END_RUNG
   RUNG wire#w3
      Contact( "hmi".model[19] )
      Move(in := 19, out1 => "currentModel")
   END_RUNG
   RUNG wire#w3
      Contact( "hmi".model[20] )
      Move(in := 20, out1 => "currentModel")
   END_RUNG
   RUNG wire#w3
      Contact( "hmi".model[21] )
      Move(in := 21, out1 => "currentModel")
   END_RUNG
   RUNG wire#w3
      Contact( "hmi".model[22] )
      Move(in := 22, out1 => "currentModel")
   END_RUNG
   RUNG wire#w3
      Contact( "hmi".model[23] )
      Move(in := 23, out1 => "currentModel")
   END_RUNG
   RUNG wire#w3
      Contact( "hmi".model[24] )
      Move(in := 24, out1 => "currentModel")
   END_RUNG
   RUNG wire#w3
      Contact( "hmi".model[25] )
      Move(in := 25, out1 => "currentModel")
   END_RUNG
   RUNG wire#w3
      Contact( "hmi".model[26] )
      Move(in := 26, out1 => "currentModel")
   END_RUNG
   RUNG wire#w3
      Contact( "hmi".model[27] )
      Move(in := 27, out1 => "currentModel")
   END_RUNG
   RUNG wire#w3
      Contact( "hmi".model[28] )
      Move(in := 28, out1 => "currentModel")
   END_RUNG
   RUNG wire#w3
      Contact( "hmi".model[29] )
      Move(in := 29, out1 => "currentModel")
   END_RUNG
   RUNG wire#w3
      Contact( "hmi".model[30] )
      Move(in := 30, out1 => "currentModel")
   END_RUNG
   RUNG wire#w3
      Contact( "hmi".model[31] )
      Move(in := 31, out1 => "currentModel")
   END_RUNG
   RUNG wire#w3
      Contact( "hmi".model[32] )
      Move(in := 32, out1 => "currentModel")
   END_RUNG
   // the same network as SCL:
   "modelChangePermit" := (NOT "outputs".activeAlarm OR ((0 = "alarm0") AND (512 = "alarm1") AND (0 = "alarm2")) OR "LOG1") AND (("currentStep" = 0) OR ("currentStep" = 1));
   IF "modelChangePermit" AND "hmi".model[1] THEN "currentModel" := 1; END_IF;
   IF "modelChangePermit" AND "hmi".model[2] THEN "currentModel" := 2; END_IF;
   IF "modelChangePermit" AND "hmi".model[3] THEN "currentModel" := 3; END_IF;
   IF "modelChangePermit" AND "hmi".model[4] THEN "currentModel" := 4; END_IF;
   IF "modelChangePermit" AND "hmi".model[5] THEN "currentModel" := 5; END_IF;
   IF "modelChangePermit" AND "hmi".model[6] THEN "currentModel" := 6; END_IF;
   IF "modelChangePermit" AND "hmi".model[7] THEN "currentModel" := 7; END_IF;
   IF "modelChangePermit" AND "hmi".model[8] THEN "currentModel" := 8; END_IF;
   IF "modelChangePermit" AND "hmi".model[9] THEN "currentModel" := 9; END_IF;
   IF "modelChangePermit" AND "hmi".model[10] THEN "currentModel" := 10; END_IF;
   IF "modelChangePermit" AND "hmi".model[11] THEN "currentModel" := 11; END_IF;
   IF "modelChangePermit" AND "hmi".model[12] THEN "currentModel" := 12; END_IF;
   IF "modelChangePermit" AND "hmi".model[13] THEN "currentModel" := 13; END_IF;
   IF "modelChangePermit" AND "hmi".model[14] THEN "currentModel" := 14; END_IF;
   IF "modelChangePermit" AND "hmi".model[15] THEN "currentModel" := 15; END_IF;
   IF "modelChangePermit" AND "hmi".model[16] THEN "currentModel" := 16; END_IF;
   IF "modelChangePermit" AND "hmi".model[15] THEN "currentModel" := 15; END_IF;
   IF "modelChangePermit" AND "hmi".model[17] THEN "currentModel" := 17; END_IF;
   IF "modelChangePermit" AND "hmi".model[18] THEN "currentModel" := 18; END_IF;
   IF "modelChangePermit" AND "hmi".model[19] THEN "currentModel" := 19; END_IF;
   IF "modelChangePermit" AND "hmi".model[20] THEN "currentModel" := 20; END_IF;
   IF "modelChangePermit" AND "hmi".model[21] THEN "currentModel" := 21; END_IF;
   IF "modelChangePermit" AND "hmi".model[22] THEN "currentModel" := 22; END_IF;
   IF "modelChangePermit" AND "hmi".model[23] THEN "currentModel" := 23; END_IF;
   IF "modelChangePermit" AND "hmi".model[24] THEN "currentModel" := 24; END_IF;
   IF "modelChangePermit" AND "hmi".model[25] THEN "currentModel" := 25; END_IF;
   IF "modelChangePermit" AND "hmi".model[26] THEN "currentModel" := 26; END_IF;
   IF "modelChangePermit" AND "hmi".model[27] THEN "currentModel" := 27; END_IF;
   IF "modelChangePermit" AND "hmi".model[28] THEN "currentModel" := 28; END_IF;
   IF "modelChangePermit" AND "hmi".model[29] THEN "currentModel" := 29; END_IF;
   IF "modelChangePermit" AND "hmi".model[30] THEN "currentModel" := 30; END_IF;
   IF "modelChangePermit" AND "hmi".model[31] THEN "currentModel" := 31; END_IF;
   IF "modelChangePermit" AND "hmi".model[32] THEN "currentModel" := 32; END_IF;
END_REGION

REGION Network 3: GAP LEADER HMI MODE
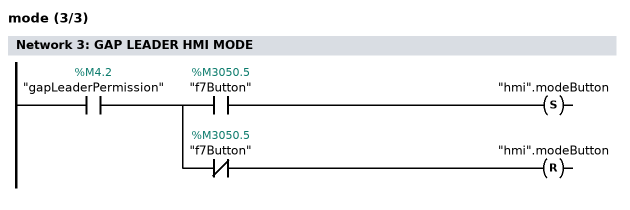
   RUNG wire#powerrail
      Contact( "gapLeaderPermission" )
      wire#w1
      Contact( "f7Button" )
      S_Coil( "hmi".modeButton )
   END_RUNG
   RUNG wire#w1
      I_Contact( "f7Button" )
      R_Coil( "hmi".modeButton )
   END_RUNG
   // the same network as SCL:
   IF "gapLeaderPermission" AND "f7Button" THEN "hmi".modeButton := TRUE; END_IF;
   IF "gapLeaderPermission" AND NOT "f7Button" THEN "hmi".modeButton := FALSE; END_IF;
END_REGION
END_FUNCTION

FUNCTION "miscelaneous" : Void   // FC5, LAD
{ S7_Optimized_Access := 'TRUE' }
VERSION : 0.1
// stored: AutoNumber true, IsIECCheckEnabled false, SetENOAutomatically false, UDAEnableTagReadback false
   VAR_TEMP
      INTERMITENTE : Bool;
      RESETEADO : Bool;
      RESULT_2 : UInt;
      Result_3 : Int;
   END_VAR
   VAR_TEMP   // added for the SCL form of the ladder/FBD networks
      _w1 : Bool;
      _w2 : Bool;
      _w3 : Bool;
      _w4 : Bool;
   END_VAR
BEGIN

REGION Network 1: HMI OPTIONS BUTTON SHUTOFF
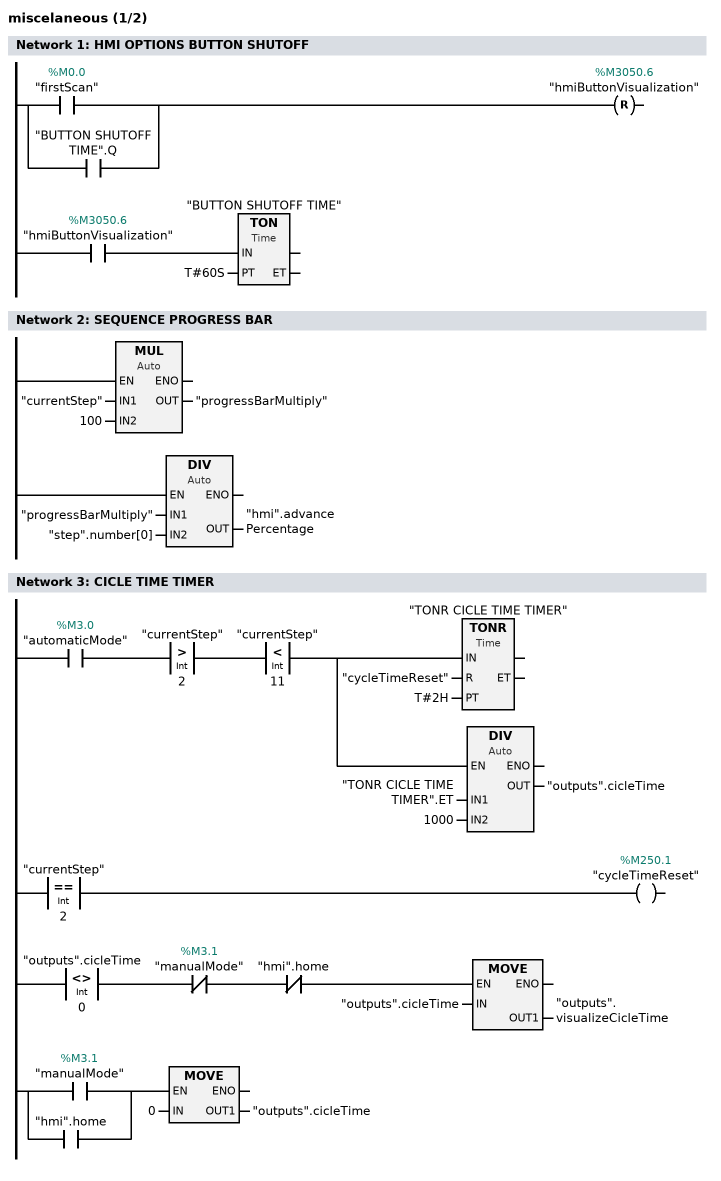
   RUNG wire#powerrail
      Contact( "firstScan" )
      wire#w1
      R_Coil( "hmiButtonVisualization" )
   END_RUNG
   RUNG wire#powerrail
      Contact( "BUTTON SHUTOFF TIME".Q )
   END_RUNG wire#w1
   RUNG wire#powerrail
      Contact( "hmiButtonVisualization" )
      { S7_Templates := "time_type := Time" } "BUTTON SHUTOFF TIME".TON(pt := T#60S, et =>)
   END_RUNG
   // the same network as SCL:
   IF "firstScan" OR "BUTTON SHUTOFF TIME".Q THEN "hmiButtonVisualization" := FALSE; END_IF;
   "BUTTON SHUTOFF TIME".TON(IN := "hmiButtonVisualization", PT := T#60S);
END_REGION

REGION Network 2: SEQUENCE PROGRESS BAR
   RUNG wire#powerrail
      Mul(in1 := "currentStep", in2 := 100, out => "progressBarMultiply")
   END_RUNG
   RUNG wire#powerrail
      Div(in1 := "progressBarMultiply", in2 := "step".number[0], out => "hmi".advancePercentage)
   END_RUNG
   // the same network as SCL:
   "progressBarMultiply" := "currentStep" * 100;
   "hmi".advancePercentage := "progressBarMultiply" / "step".number[0];
END_REGION

REGION Network 3: CICLE TIME TIMER
   RUNG wire#powerrail
      Contact( "automaticMode" )
      { S7_Templates := "SrcType := Int" } GT_Contact(in1 := "currentStep", in2 := 2)
      { S7_Templates := "SrcType := Int" } LT_Contact(in1 := "currentStep", in2 := 11)
      wire#w1
      { S7_Templates := "time_type := Time" } "TONR CICLE TIME TIMER".TONR(r := "cycleTimeReset", pt := T#2H, et =>)
   END_RUNG
   RUNG wire#w1
      Div(in1 := "TONR CICLE TIME TIMER".ET, in2 := 1000, out => "outputs".cicleTime)
   END_RUNG
   RUNG wire#powerrail
      { S7_Templates := "SrcType := Int" } EQ_Contact(in1 := "currentStep", in2 := 2)
      Coil( "cycleTimeReset" )
   END_RUNG
   RUNG wire#powerrail
      { S7_Templates := "SrcType := Int" } NE_Contact(in1 := "outputs".cicleTime, in2 := 0)
      I_Contact( "manualMode" )
      I_Contact( "hmi".home )
      Move(in := "outputs".cicleTime, out1 => "outputs".visualizeCicleTime)
   END_RUNG
   RUNG wire#powerrail
      Contact( "manualMode" )
      wire#w2
      Move(in := 0, out1 => "outputs".cicleTime)
   END_RUNG
   RUNG wire#powerrail
      Contact( "hmi".home )
   END_RUNG wire#w2
   // the same network as SCL:
   #_w1 := "automaticMode" AND ("currentStep" > 2) AND ("currentStep" < 11);
   "TONR CICLE TIME TIMER".TONR(IN := #_w1, R := "cycleTimeReset", PT := T#2H);
   IF #_w1 THEN "outputs".cicleTime := "TONR CICLE TIME TIMER".ET / 1000; END_IF;
   "cycleTimeReset" := "currentStep" = 2;
   IF ("outputs".cicleTime <> 0) AND NOT "manualMode" AND NOT "hmi".home THEN
       "outputs".visualizeCicleTime := "outputs".cicleTime;
   END_IF;
   IF "manualMode" OR "hmi".home THEN "outputs".cicleTime := 0; END_IF;
END_REGION

REGION Network 4: STEP CHANGE TIMER
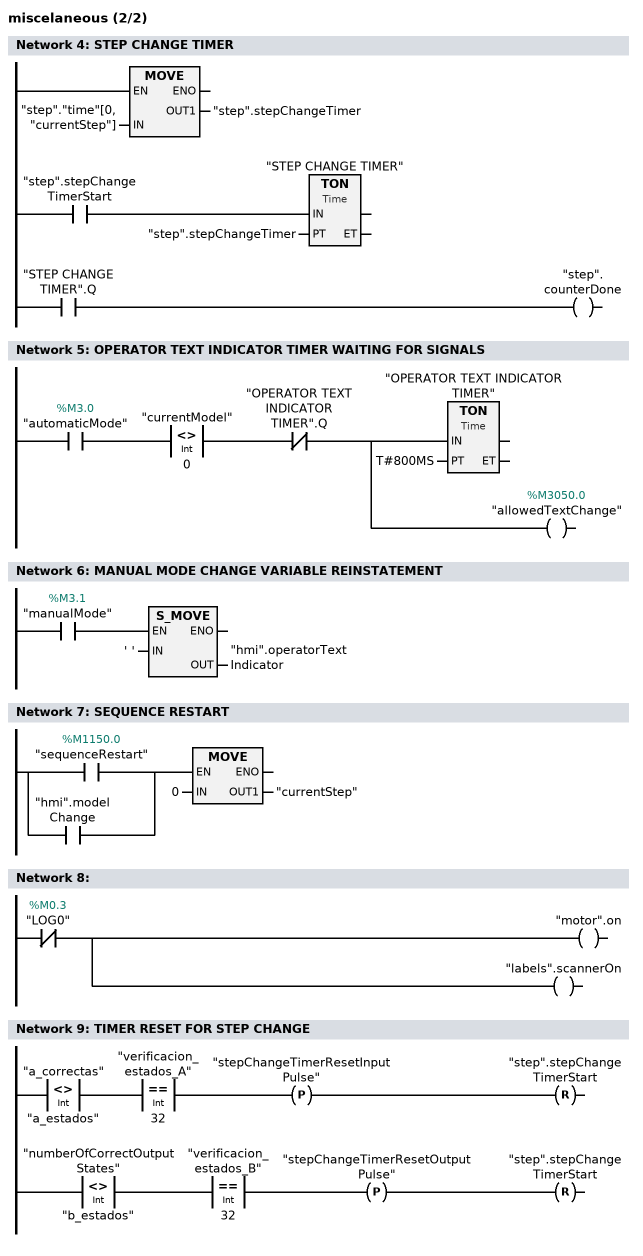
   RUNG wire#powerrail
      Move(in := "step"."time"[0, "currentStep"], out1 => "step".stepChangeTimer)
   END_RUNG
   RUNG wire#powerrail
      Contact( "step".stepChangeTimerStart )
      { S7_Templates := "time_type := Time" } "STEP CHANGE TIMER".TON(pt := "step".stepChangeTimer, et =>)
   END_RUNG
   RUNG wire#powerrail
      Contact( "STEP CHANGE TIMER".Q )
      Coil( "step".counterDone )
   END_RUNG
   // the same network as SCL:
   "step".stepChangeTimer := "step"."time"[0, "currentStep"];
   "STEP CHANGE TIMER".TON(IN := "step".stepChangeTimerStart, PT := "step".stepChangeTimer);
   "step".counterDone := "STEP CHANGE TIMER".Q;
END_REGION

REGION Network 5: OPERATOR TEXT INDICATOR TIMER WAITING FOR SIGNALS
   RUNG wire#powerrail
      Contact( "automaticMode" )
      { S7_Templates := "SrcType := Int" } NE_Contact(in1 := "currentModel", in2 := 0)
      I_Contact( "OPERATOR TEXT INDICATOR TIMER".Q )
      wire#w1
      { S7_Templates := "time_type := Time" } "OPERATOR TEXT INDICATOR TIMER".TON(pt := T#800MS, et =>)
   END_RUNG
   RUNG wire#w1
      Coil( "allowedTextChange" )
   END_RUNG
   // the same network as SCL:
   #_w1 := "automaticMode" AND ("currentModel" <> 0) AND NOT "OPERATOR TEXT INDICATOR TIMER".Q;
   "OPERATOR TEXT INDICATOR TIMER".TON(IN := #_w1, PT := T#800MS);
   "allowedTextChange" := #_w1;
END_REGION

REGION Network 6: MANUAL MODE CHANGE VARIABLE REINSTATEMENT
   RUNG wire#powerrail
      Contact( "manualMode" )
      S_Move(in := ' ', out => "hmi".operatorTextIndicator)
   END_RUNG
   // the same network as SCL:
   IF "manualMode" THEN "hmi".operatorTextIndicator := ' '; END_IF;
END_REGION

REGION Network 7: SEQUENCE RESTART
   RUNG wire#powerrail
      Contact( "sequenceRestart" )
      wire#w1
      Move(in := 0, out1 => "currentStep")
   END_RUNG
   RUNG wire#powerrail
      Contact( "hmi".modelChange )
   END_RUNG wire#w1
   // the same network as SCL:
   IF "sequenceRestart" OR "hmi".modelChange THEN "currentStep" := 0; END_IF;
END_REGION

REGION Network 8
   RUNG wire#powerrail
      I_Contact( "LOG0" )
      wire#w1
      Coil( "motor".on )
   END_RUNG
   RUNG wire#w1
      Coil( "labels".scannerOn )
   END_RUNG
   // the same network as SCL:
   "motor".on := NOT "LOG0";
   "labels".scannerOn := NOT "LOG0";
END_REGION

REGION Network 9: TIMER RESET FOR STEP CHANGE
   RUNG wire#powerrail
      { S7_Templates := "SrcType := Int" } NE_Contact(in1 := "a_correctas", in2 := "a_estados")
      { S7_Templates := "SrcType := Int" } EQ_Contact(in1 := "verificacion_estados_A", in2 := 32)
      P_Trig( "stepChangeTimerResetInputPulse" )
      R_Coil( "step".stepChangeTimerStart )
   END_RUNG
   RUNG wire#powerrail
      { S7_Templates := "SrcType := Int" } NE_Contact(in1 := "numberOfCorrectOutputStates", in2 := "b_estados")
      { S7_Templates := "SrcType := Int" } EQ_Contact(in1 := "verificacion_estados_B", in2 := 32)
      P_Trig( "stepChangeTimerResetOutputPulse" )
      R_Coil( "step".stepChangeTimerStart )
   END_RUNG
   // the same network as SCL:
   #_w1 := ("a_correctas" <> "a_estados") AND ("verificacion_estados_A" = 32);
   #_w2 := #_w1 AND NOT "stepChangeTimerResetInputPulse";   // rising edge
   "stepChangeTimerResetInputPulse" := #_w1;
   IF #_w2 THEN "step".stepChangeTimerStart := FALSE; END_IF;
   #_w3 := ("numberOfCorrectOutputStates" <> "b_estados") AND ("verificacion_estados_B" = 32);
   #_w4 := #_w3 AND NOT "stepChangeTimerResetOutputPulse";   // rising edge
   "stepChangeTimerResetOutputPulse" := #_w3;
   IF #_w4 THEN "step".stepChangeTimerStart := FALSE; END_IF;
END_REGION
END_FUNCTION

FUNCTION "modifyRecipe" : Void   // FC6, LAD
{ S7_Optimized_Access := 'TRUE' }
VERSION : 0.1
// stored: AutoNumber true, IsIECCheckEnabled false, SetENOAutomatically false, UDAEnableTagReadback false
   VAR_TEMP   // added for the SCL form of the ladder/FBD networks
      _w1 : Bool;
      _w2 : Bool;
   END_VAR
BEGIN

REGION Network 1: ERASE A STEP
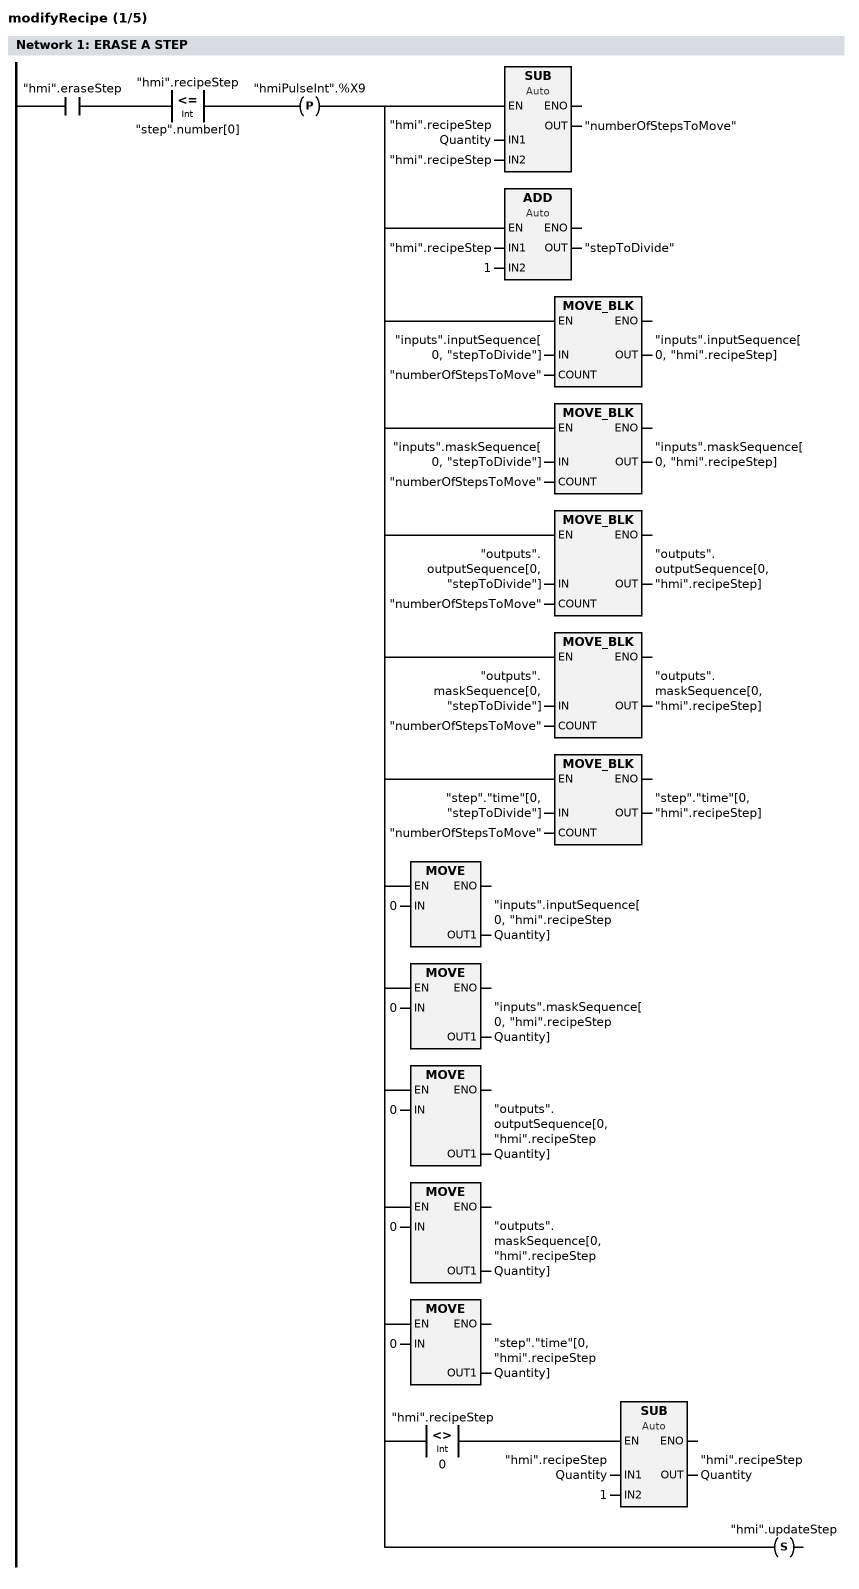
   #_w1 := "hmi".eraseStep AND ("hmi".recipeStep <= "step".number[0]);
   #_w2 := #_w1 AND NOT "hmiPulseInt".%X9;   // rising edge
   "hmiPulseInt".%X9 := #_w1;
   IF #_w2 THEN
       "numberOfStepsToMove" := "hmi".recipeStepQuantity - "hmi".recipeStep;
       "stepToDivide" := "hmi".recipeStep + 1;
       MOVE_BLK(IN := "inputs".inputSequence[0, "stepToDivide"],
                COUNT := "numberOfStepsToMove",
                OUT => "inputs".inputSequence[0, "hmi".recipeStep]);
       MOVE_BLK(IN := "inputs".maskSequence[0, "stepToDivide"],
                COUNT := "numberOfStepsToMove",
                OUT => "inputs".maskSequence[0, "hmi".recipeStep]);
       MOVE_BLK(IN := "outputs".outputSequence[0, "stepToDivide"],
                COUNT := "numberOfStepsToMove",
                OUT => "outputs".outputSequence[0, "hmi".recipeStep]);
       MOVE_BLK(IN := "outputs".maskSequence[0, "stepToDivide"],
                COUNT := "numberOfStepsToMove",
                OUT => "outputs".maskSequence[0, "hmi".recipeStep]);
       MOVE_BLK(IN := "step"."time"[0, "stepToDivide"],
                COUNT := "numberOfStepsToMove",
                OUT => "step"."time"[0, "hmi".recipeStep]);
       "inputs".inputSequence[0, "hmi".recipeStepQuantity] := 0;
       "inputs".maskSequence[0, "hmi".recipeStepQuantity] := 0;
       "outputs".outputSequence[0, "hmi".recipeStepQuantity] := 0;
       "outputs".maskSequence[0, "hmi".recipeStepQuantity] := 0;
       "step"."time"[0, "hmi".recipeStepQuantity] := 0;
   END_IF;
   IF #_w2 AND ("hmi".recipeStep <> 0) THEN "hmi".recipeStepQuantity := "hmi".recipeStepQuantity - 1; END_IF;
   IF #_w2 THEN "hmi".updateStep := TRUE; END_IF;
END_REGION

